    CONST robtarget p14641:= [[1510.9571216135703, 63.37345761549072, 1006.500033578516], [0, 0, 1, 0], [0, 0, 0, 0], [9E9, 9E9, 9E9, 9E9, 9E9, 9E9]];
    CONST robtarget p14642:= [[1511.1184630222722, 63.35487120853786, 1006.500033578516], [0, 0, 1, 0], [0, 0, 0, 0], [9E9, 9E9, 9E9, 9E9, 9E9, 9E9]];
    CONST robtarget p14643:= [[1511.1919380294153, 63.341381931287984, 1006.500033578516], [0, 0, 1, 0], [0, 0, 0, 0], [9E9, 9E9, 9E9, 9E9, 9E9, 9E9]];
    CONST robtarget p14644:= [[1512.026838057439, 63.17846774539392, 1006.500033578516], [0, 0, 1, 0], [0, 0, 0, 0], [9E9, 9E9, 9E9, 9E9, 9E9, 9E9]];
    CONST robtarget p14645:= [[1512.5585207158877, 63.05117882240624, 1006.500033578516], [0, 0, 1, 0], [0, 0, 0, 0], [9E9, 9E9, 9E9, 9E9, 9E9, 9E9]];
    CONST robtarget p14646:= [[1512.9152156348257, 62.99334195486536, 1006.500033578516], [0, 0, 1, 0], [0, 0, 0, 0], [9E9, 9E9, 9E9, 9E9, 9E9, 9E9]];
    CONST robtarget p14647:= [[1513.798506951844, 62.783709162407874, 1006.500033578516], [0, 0, 1, 0], [0, 0, 0, 0], [9E9, 9E9, 9E9, 9E9, 9E9, 9E9]];
    CONST robtarget p14648:= [[1514.847567863613, 62.563530246518, 1006.500033578516], [0, 0, 1, 0], [0, 0, 0, 0], [9E9, 9E9, 9E9, 9E9, 9E9, 9E9]];
    CONST robtarget p14649:= [[1515.255096833937, 62.462945925381334, 1006.500033578516], [0, 0, 1, 0], [0, 0, 0, 0], [9E9, 9E9, 9E9, 9E9, 9E9, 9E9]];
    CONST robtarget p14650:= [[1515.509041751135, 62.41476108124637, 1006.500033578516], [0, 0, 1, 0], [0, 0, 0, 0], [9E9, 9E9, 9E9, 9E9, 9E9, 9E9]];
    CONST robtarget p14651:= [[1515.8348657437182, 62.34037513585322, 1006.500033578516], [0, 0, 1, 0], [0, 0, 0, 0], [9E9, 9E9, 9E9, 9E9, 9E9, 9E9]];
    CONST robtarget p14652:= [[1516.3628032758625, 62.21258930958216, 1006.500033578516], [0, 0, 1, 0], [0, 0, 0, 0], [9E9, 9E9, 9E9, 9E9, 9E9, 9E9]];
    CONST robtarget p14653:= [[1516.8558086004887, 62.054342846622134, 1006.500033578516], [0, 0, 1, 0], [0, 0, 0, 0], [9E9, 9E9, 9E9, 9E9, 9E9, 9E9]];
    CONST robtarget p14654:= [[1516.94184995351, 62.01985911324756, 1006.500033578516], [0, 0, 1, 0], [0, 0, 0, 0], [9E9, 9E9, 9E9, 9E9, 9E9, 9E9]];
    CONST robtarget p14655:= [[1517.8260139593945, 61.7655492376807, 1006.500033578516], [0, 0, 1, 0], [0, 0, 0, 0], [9E9, 9E9, 9E9, 9E9, 9E9, 9E9]];
    CONST robtarget p14656:= [[1518.3959985979216, 61.59972849280017, 1006.500033578516], [0, 0, 1, 0], [0, 0, 0, 0], [9E9, 9E9, 9E9, 9E9, 9E9, 9E9]];
    CONST robtarget p14657:= [[1519.0877750129548, 61.40495027580202, 1006.500033578516], [0, 0, 1, 0], [0, 0, 0, 0], [9E9, 9E9, 9E9, 9E9, 9E9, 9E9]];
    CONST robtarget p14658:= [[1519.4220256911422, 61.30068815369448, 1006.500033578516], [0, 0, 1, 0], [0, 0, 0, 0], [9E9, 9E9, 9E9, 9E9, 9E9, 9E9]];
    CONST robtarget p14659:= [[1520.4546810078716, 60.9628761084728, 1006.500033578516], [0, 0, 1, 0], [0, 0, 0, 0], [9E9, 9E9, 9E9, 9E9, 9E9, 9E9]];
    CONST robtarget p14660:= [[1520.7208420853615, 60.899099294826286, 1006.500033578516], [0, 0, 1, 0], [0, 0, 0, 0], [9E9, 9E9, 9E9, 9E9, 9E9, 9E9]];
    CONST robtarget p14661:= [[1520.9944154401092, 60.79050565777585, 1006.500033578516], [0, 0, 1, 0], [0, 0, 0, 0], [9E9, 9E9, 9E9, 9E9, 9E9, 9E9]];
    CONST robtarget p14662:= [[1521.468460467742, 60.619702144143545, 1006.500033578516], [0, 0, 1, 0], [0, 0, 0, 0], [9E9, 9E9, 9E9, 9E9, 9E9, 9E9]];
    CONST robtarget p14663:= [[1522.0539891001142, 60.40291207086237, 1006.500033578516], [0, 0, 1, 0], [0, 0, 0, 0], [9E9, 9E9, 9E9, 9E9, 9E9, 9E9]];
    CONST robtarget p14664:= [[1522.7235250206843, 60.13765981750545, 1006.500033578516], [0, 0, 1, 0], [0, 0, 0, 0], [9E9, 9E9, 9E9, 9E9, 9E9, 9E9]];
    CONST robtarget p14665:= [[1522.7540810701935, 60.12646280502547, 1006.500033578516], [0, 0, 1, 0], [0, 0, 0, 0], [9E9, 9E9, 9E9, 9E9, 9E9, 9E9]];
    CONST robtarget p14666:= [[1522.977172790825, 60.0450909611216, 1006.500033578516], [0, 0, 1, 0], [0, 0, 0, 0], [9E9, 9E9, 9E9, 9E9, 9E9, 9E9]];
    CONST robtarget p14667:= [[1523.8573489774064, 59.71048583629785, 1006.500033578516], [0, 0, 1, 0], [0, 0, 0, 0], [9E9, 9E9, 9E9, 9E9, 9E9, 9E9]];
    CONST robtarget p14668:= [[1524.305158114966, 59.53535137429769, 1006.500033578516], [0, 0, 1, 0], [0, 0, 0, 0], [9E9, 9E9, 9E9, 9E9, 9E9, 9E9]];
    CONST robtarget p14669:= [[1524.656610079094, 59.40530950563833, 1006.500033578516], [0, 0, 1, 0], [0, 0, 0, 0], [9E9, 9E9, 9E9, 9E9, 9E9, 9E9]];
    CONST robtarget p14670:= [[1525.149298617828, 59.17779911458156, 1006.500033578516], [0, 0, 1, 0], [0, 0, 0, 0], [9E9, 9E9, 9E9, 9E9, 9E9, 9E9]];
    CONST robtarget p14671:= [[1525.7575127352557, 58.87613102467979, 1006.500033578516], [0, 0, 1, 0], [0, 0, 0, 0], [9E9, 9E9, 9E9, 9E9, 9E9, 9E9]];
    CONST robtarget p14672:= [[1526.170972481238, 58.714980753068446, 1006.500033578516], [0, 0, 1, 0], [0, 0, 0, 0], [9E9, 9E9, 9E9, 9E9, 9E9, 9E9]];
    CONST robtarget p14673:= [[1526.7257950856722, 58.46470075930664, 1006.500033578516], [0, 0, 1, 0], [0, 0, 0, 0], [9E9, 9E9, 9E9, 9E9, 9E9, 9E9]];
    CONST robtarget p14674:= [[1527.3077094242446, 58.20997178842184, 1006.500033578516], [0, 0, 1, 0], [0, 0, 0, 0], [9E9, 9E9, 9E9, 9E9, 9E9, 9E9]];
    CONST robtarget p14675:= [[1527.6845666037234, 58.0161366438124, 1006.500033578516], [0, 0, 1, 0], [0, 0, 0, 0], [9E9, 9E9, 9E9, 9E9, 9E9, 9E9]];
    CONST robtarget p14676:= [[1527.8326061398718, 57.948812745233525, 1006.500033578516], [0, 0, 1, 0], [0, 0, 0, 0], [9E9, 9E9, 9E9, 9E9, 9E9, 9E9]];
    CONST robtarget p14677:= [[1528.3321808852675, 57.69325378961487, 1006.500033578516], [0, 0, 1, 0], [0, 0, 0, 0], [9E9, 9E9, 9E9, 9E9, 9E9, 9E9]];
    CONST robtarget p14678:= [[1528.403927309375, 57.65748391653119, 1006.500033578516], [0, 0, 1, 0], [0, 0, 0, 0], [9E9, 9E9, 9E9, 9E9, 9E9, 9E9]];
    CONST robtarget p14679:= [[1528.9869187812067, 57.39394460057444, 1006.500033578516], [0, 0, 1, 0], [0, 0, 0, 0], [9E9, 9E9, 9E9, 9E9, 9E9, 9E9]];
    CONST robtarget p14680:= [[1529.2613805009244, 57.26779957940987, 1006.500033578516], [0, 0, 1, 0], [0, 0, 0, 0], [9E9, 9E9, 9E9, 9E9, 9E9, 9E9]];
    CONST robtarget p14681:= [[1529.6697738066682, 57.06843620345721, 1006.500033578516], [0, 0, 1, 0], [0, 0, 0, 0], [9E9, 9E9, 9E9, 9E9, 9E9, 9E9]];
    CONST robtarget p14682:= [[1530.2856563586133, 56.72445722365994, 1006.500033578516], [0, 0, 1, 0], [0, 0, 0, 0], [9E9, 9E9, 9E9, 9E9, 9E9, 9E9]];
    CONST robtarget p14683:= [[1530.8126991827496, 56.4341660345891, 1006.500033578516], [0, 0, 1, 0], [0, 0, 0, 0], [9E9, 9E9, 9E9, 9E9, 9E9, 9E9]];
    CONST robtarget p14684:= [[1530.9029259654756, 56.3783277374728, 1006.500033578516], [0, 0, 1, 0], [0, 0, 0, 0], [9E9, 9E9, 9E9, 9E9, 9E9, 9E9]];
    CONST robtarget p14685:= [[1531.0054963877374, 56.315172306385094, 1006.500033578516], [0, 0, 1, 0], [0, 0, 0, 0], [9E9, 9E9, 9E9, 9E9, 9E9, 9E9]];
    CONST robtarget p14686:= [[1531.3939612691959, 56.09683858981346, 1006.500033578516], [0, 0, 1, 0], [0, 0, 0, 0], [9E9, 9E9, 9E9, 9E9, 9E9, 9E9]];
    CONST robtarget p14687:= [[1531.8623727083182, 55.83685599433868, 1006.500033578516], [0, 0, 1, 0], [0, 0, 0, 0], [9E9, 9E9, 9E9, 9E9, 9E9, 9E9]];
    CONST robtarget p14688:= [[1532.024440070901, 55.73722495097826, 1006.500033578516], [0, 0, 1, 0], [0, 0, 0, 0], [9E9, 9E9, 9E9, 9E9, 9E9, 9E9]];
    CONST robtarget p14689:= [[1532.7201519563368, 55.36777082129741, 1006.500033578516], [0, 0, 1, 0], [0, 0, 0, 0], [9E9, 9E9, 9E9, 9E9, 9E9, 9E9]];
    CONST robtarget p14690:= [[1533.2451221887477, 55.05705588289027, 1006.500033578516], [0, 0, 1, 0], [0, 0, 0, 0], [9E9, 9E9, 9E9, 9E9, 9E9, 9E9]];
    CONST robtarget p14691:= [[1533.6846313226854, 54.805458357707266, 1006.500033578516], [0, 0, 1, 0], [0, 0, 0, 0], [9E9, 9E9, 9E9, 9E9, 9E9, 9E9]];
    CONST robtarget p14692:= [[1533.8934584959652, 54.65278530648348, 1006.500033578516], [0, 0, 1, 0], [0, 0, 0, 0], [9E9, 9E9, 9E9, 9E9, 9E9, 9E9]];
    CONST robtarget p14693:= [[1534.2116287991314, 54.4123880238884, 1006.500033578516], [0, 0, 1, 0], [0, 0, 0, 0], [9E9, 9E9, 9E9, 9E9, 9E9, 9E9]];
    CONST robtarget p14694:= [[1534.6901098946857, 54.118222023287345, 1006.500033578516], [0, 0, 1, 0], [0, 0, 0, 0], [9E9, 9E9, 9E9, 9E9, 9E9, 9E9]];
    CONST robtarget p14695:= [[1535.3882444304677, 53.67964368227618, 1006.500033578516], [0, 0, 1, 0], [0, 0, 0, 0], [9E9, 9E9, 9E9, 9E9, 9E9, 9E9]];
    CONST robtarget p14696:= [[1535.6440065674608, 53.48641652408345, 1006.500033578516], [0, 0, 1, 0], [0, 0, 0, 0], [9E9, 9E9, 9E9, 9E9, 9E9, 9E9]];
    CONST robtarget p14697:= [[1536.2093768314423, 53.097910660736204, 1006.500033578516], [0, 0, 1, 0], [0, 0, 0, 0], [9E9, 9E9, 9E9, 9E9, 9E9, 9E9]];
    CONST robtarget p14698:= [[1536.9779076559207, 52.624035474973724, 1006.500033578516], [0, 0, 1, 0], [0, 0, 0, 0], [9E9, 9E9, 9E9, 9E9, 9E9, 9E9]];
    CONST robtarget p14699:= [[1537.4393405989101, 52.32171516144058, 1006.500033578516], [0, 0, 1, 0], [0, 0, 0, 0], [9E9, 9E9, 9E9, 9E9, 9E9, 9E9]];
    CONST robtarget p14700:= [[1537.952006745379, 51.91517388024164, 1006.500033578516], [0, 0, 1, 0], [0, 0, 0, 0], [9E9, 9E9, 9E9, 9E9, 9E9, 9E9]];
    CONST robtarget p14701:= [[1538.2226229328674, 51.700360577582046, 1006.500033578516], [0, 0, 1, 0], [0, 0, 0, 0], [9E9, 9E9, 9E9, 9E9, 9E9, 9E9]];
    CONST robtarget p14702:= [[1538.5500075167402, 51.46408461899675, 1006.500033578516], [0, 0, 1, 0], [0, 0, 0, 0], [9E9, 9E9, 9E9, 9E9, 9E9, 9E9]];
    CONST robtarget p14703:= [[1538.9225032761597, 51.18184185491022, 1006.500033578516], [0, 0, 1, 0], [0, 0, 0, 0], [9E9, 9E9, 9E9, 9E9, 9E9, 9E9]];
    CONST robtarget p14704:= [[1539.2375324072243, 50.939131502791724, 1006.500033578516], [0, 0, 1, 0], [0, 0, 0, 0], [9E9, 9E9, 9E9, 9E9, 9E9, 9E9]];
    CONST robtarget p14705:= [[1540.1829191616407, 50.145246062498, 1006.500033578516], [0, 0, 1, 0], [0, 0, 0, 0], [9E9, 9E9, 9E9, 9E9, 9E9, 9E9]];
    CONST robtarget p14706:= [[1540.6342645888235, 49.82479613541888, 1006.500033578516], [0, 0, 1, 0], [0, 0, 0, 0], [9E9, 9E9, 9E9, 9E9, 9E9, 9E9]];
    CONST robtarget p14707:= [[1541.3997951640697, 49.20201413735353, 1006.500033578516], [0, 0, 1, 0], [0, 0, 0, 0], [9E9, 9E9, 9E9, 9E9, 9E9, 9E9]];
    CONST robtarget p14708:= [[1542.2802015710938, 48.44291913123219, 1006.500033578516], [0, 0, 1, 0], [0, 0, 0, 0], [9E9, 9E9, 9E9, 9E9, 9E9, 9E9]];
    CONST robtarget p14709:= [[1542.848436210057, 47.911154253194894, 1006.500033578516], [0, 0, 1, 0], [0, 0, 0, 0], [9E9, 9E9, 9E9, 9E9, 9E9, 9E9]];
    CONST robtarget p14710:= [[1543.249750681818, 47.58041096004163, 1006.500033578516], [0, 0, 1, 0], [0, 0, 0, 0], [9E9, 9E9, 9E9, 9E9, 9E9, 9E9]];
    CONST robtarget p14711:= [[1543.8613961148844, 46.98941101413523, 1006.500033578516], [0, 0, 1, 0], [0, 0, 0, 0], [9E9, 9E9, 9E9, 9E9, 9E9, 9E9]];
    CONST robtarget p14712:= [[1544.0446499071509, 46.83874137102008, 1006.500033578516], [0, 0, 1, 0], [0, 0, 0, 0], [9E9, 9E9, 9E9, 9E9, 9E9, 9E9]];
    CONST robtarget p14713:= [[1544.2953989022335, 46.61563060487386, 1006.500033578516], [0, 0, 1, 0], [0, 0, 0, 0], [9E9, 9E9, 9E9, 9E9, 9E9, 9E9]];
    CONST robtarget p14714:= [[1544.54804056772, 46.38574176255722, 1006.500033578516], [0, 0, 1, 0], [0, 0, 0, 0], [9E9, 9E9, 9E9, 9E9, 9E9, 9E9]];
    CONST robtarget p14715:= [[1544.635189922801, 46.31124549330636, 1006.500033578516], [0, 0, 1, 0], [0, 0, 0, 0], [9E9, 9E9, 9E9, 9E9, 9E9, 9E9]];
    CONST robtarget p14716:= [[1545.4540333634932, 45.48335179072561, 1006.500033578516], [0, 0, 1, 0], [0, 0, 0, 0], [9E9, 9E9, 9E9, 9E9, 9E9, 9E9]];
    CONST robtarget p14717:= [[1545.7644585194985, 45.10437831876281, 1006.500033578516], [0, 0, 1, 0], [0, 0, 0, 0], [9E9, 9E9, 9E9, 9E9, 9E9, 9E9]];
    CONST robtarget p14718:= [[1546.0127018950527, 44.843745114856446, 1006.500033578516], [0, 0, 1, 0], [0, 0, 0, 0], [9E9, 9E9, 9E9, 9E9, 9E9, 9E9]];
    CONST robtarget p14719:= [[1546.7740572911337, 44.03270232293215, 1006.500033578516], [0, 0, 1, 0], [0, 0, 0, 0], [9E9, 9E9, 9E9, 9E9, 9E9, 9E9]];
    CONST robtarget p14720:= [[1547.0970360263204, 43.759023791525095, 1006.500033578516], [0, 0, 1, 0], [0, 0, 0, 0], [9E9, 9E9, 9E9, 9E9, 9E9, 9E9]];
    CONST robtarget p14721:= [[1547.2985281571125, 43.556821645131976, 1006.500033578516], [0, 0, 1, 0], [0, 0, 0, 0], [9E9, 9E9, 9E9, 9E9, 9E9, 9E9]];
    CONST robtarget p14722:= [[1547.5784264326533, 43.24559099443002, 1006.500033578516], [0, 0, 1, 0], [0, 0, 0, 0], [9E9, 9E9, 9E9, 9E9, 9E9, 9E9]];
    CONST robtarget p14723:= [[1547.840639915275, 42.976910613143446, 1006.500033578516], [0, 0, 1, 0], [0, 0, 0, 0], [9E9, 9E9, 9E9, 9E9, 9E9, 9E9]];
    CONST robtarget p14724:= [[1548.5685814620201, 42.11718983212772, 1006.500033578516], [0, 0, 1, 0], [0, 0, 0, 0], [9E9, 9E9, 9E9, 9E9, 9E9, 9E9]];
    CONST robtarget p14725:= [[1549.0589016644108, 41.54224515009723, 1006.500033578516], [0, 0, 1, 0], [0, 0, 0, 0], [9E9, 9E9, 9E9, 9E9, 9E9, 9E9]];
    CONST robtarget p14726:= [[1549.1397925073998, 41.45436251768466, 1006.500033578516], [0, 0, 1, 0], [0, 0, 0, 0], [9E9, 9E9, 9E9, 9E9, 9E9, 9E9]];
    CONST robtarget p14727:= [[1549.3841406789884, 41.1427679591735, 1006.500033578516], [0, 0, 1, 0], [0, 0, 0, 0], [9E9, 9E9, 9E9, 9E9, 9E9, 9E9]];
    CONST robtarget p14728:= [[1549.5239794339052, 40.95950274767945, 1006.500033578516], [0, 0, 1, 0], [0, 0, 0, 0], [9E9, 9E9, 9E9, 9E9, 9E9, 9E9]];
    CONST robtarget p14729:= [[1549.9175539397738, 40.51438406992901, 1006.500033578516], [0, 0, 1, 0], [0, 0, 0, 0], [9E9, 9E9, 9E9, 9E9, 9E9, 9E9]];
    CONST robtarget p14730:= [[1550.3216633796537, 40.038823451018516, 1006.500033578516], [0, 0, 1, 0], [0, 0, 0, 0], [9E9, 9E9, 9E9, 9E9, 9E9, 9E9]];
    CONST robtarget p14731:= [[1550.4495787903381, 39.860864577949286, 1006.500033578516], [0, 0, 1, 0], [0, 0, 0, 0], [9E9, 9E9, 9E9, 9E9, 9E9, 9E9]];
    CONST robtarget p14732:= [[1550.6937743751787, 39.5427168649649, 1006.500033578516], [0, 0, 1, 0], [0, 0, 0, 0], [9E9, 9E9, 9E9, 9E9, 9E9, 9E9]];
    CONST robtarget p14733:= [[1551.2596416418764, 38.84732865927106, 1006.500033578516], [0, 0, 1, 0], [0, 0, 0, 0], [9E9, 9E9, 9E9, 9E9, 9E9, 9E9]];
    CONST robtarget p14734:= [[1551.6870753715048, 38.25053385446556, 1006.500033578516], [0, 0, 1, 0], [0, 0, 0, 0], [9E9, 9E9, 9E9, 9E9, 9E9, 9E9]];
    CONST robtarget p14735:= [[1551.8361490020857, 38.01625032551375, 1006.500033578516], [0, 0, 1, 0], [0, 0, 0, 0], [9E9, 9E9, 9E9, 9E9, 9E9, 9E9]];
    CONST robtarget p14736:= [[1552.322823514699, 37.36153510210862, 1006.500033578516], [0, 0, 1, 0], [0, 0, 0, 0], [9E9, 9E9, 9E9, 9E9, 9E9, 9E9]];
    CONST robtarget p14737:= [[1552.5842476544994, 36.958893981652636, 1006.500033578516], [0, 0, 1, 0], [0, 0, 0, 0], [9E9, 9E9, 9E9, 9E9, 9E9, 9E9]];
    CONST robtarget p14738:= [[1552.8616551509776, 36.5874901381969, 1006.500033578516], [0, 0, 1, 0], [0, 0, 0, 0], [9E9, 9E9, 9E9, 9E9, 9E9, 9E9]];
    CONST robtarget p14739:= [[1553.159967137924, 36.201259725787494, 1006.500033578516], [0, 0, 1, 0], [0, 0, 0, 0], [9E9, 9E9, 9E9, 9E9, 9E9, 9E9]];
    CONST robtarget p14740:= [[1553.3919006865265, 35.845938138459914, 1006.500033578516], [0, 0, 1, 0], [0, 0, 0, 0], [9E9, 9E9, 9E9, 9E9, 9E9, 9E9]];
    CONST robtarget p14741:= [[1553.4492538776192, 35.75324229238505, 1006.500033578516], [0, 0, 1, 0], [0, 0, 0, 0], [9E9, 9E9, 9E9, 9E9, 9E9, 9E9]];
    CONST robtarget p14742:= [[1553.6849733642457, 35.35776058704826, 1006.500033578516], [0, 0, 1, 0], [0, 0, 0, 0], [9E9, 9E9, 9E9, 9E9, 9E9, 9E9]];
    CONST robtarget p14743:= [[1554.0221492244746, 34.890455488715006, 1006.500033578516], [0, 0, 1, 0], [0, 0, 0, 0], [9E9, 9E9, 9E9, 9E9, 9E9, 9E9]];
    CONST robtarget p14744:= [[1554.3819330409094, 34.311998246707276, 1006.500033578516], [0, 0, 1, 0], [0, 0, 0, 0], [9E9, 9E9, 9E9, 9E9, 9E9, 9E9]];
    CONST robtarget p14745:= [[1554.7324883746796, 33.72360383375208, 1006.500033578516], [0, 0, 1, 0], [0, 0, 0, 0], [9E9, 9E9, 9E9, 9E9, 9E9, 9E9]];
    CONST robtarget p14746:= [[1554.9694331765027, 33.34150920841043, 1006.500033578516], [0, 0, 1, 0], [0, 0, 0, 0], [9E9, 9E9, 9E9, 9E9, 9E9, 9E9]];
    CONST robtarget p14747:= [[1555.0578363454322, 33.18808941710759, 1006.500033578516], [0, 0, 1, 0], [0, 0, 0, 0], [9E9, 9E9, 9E9, 9E9, 9E9, 9E9]];
    CONST robtarget p14748:= [[1555.5191903887774, 32.347242553330574, 1006.500033578516], [0, 0, 1, 0], [0, 0, 0, 0], [9E9, 9E9, 9E9, 9E9, 9E9, 9E9]];
    CONST robtarget p14749:= [[1555.899208185482, 31.751166868234478, 1006.500033578516], [0, 0, 1, 0], [0, 0, 0, 0], [9E9, 9E9, 9E9, 9E9, 9E9, 9E9]];
    CONST robtarget p14750:= [[1556.105965761014, 31.457408539315693, 1006.500033578516], [0, 0, 1, 0], [0, 0, 0, 0], [9E9, 9E9, 9E9, 9E9, 9E9, 9E9]];
    CONST robtarget p14751:= [[1556.2761023181502, 31.162061354166894, 1006.500033578516], [0, 0, 1, 0], [0, 0, 0, 0], [9E9, 9E9, 9E9, 9E9, 9E9, 9E9]];
    CONST robtarget p14752:= [[1556.420299300182, 30.87457089103094, 1006.500033578516], [0, 0, 1, 0], [0, 0, 0, 0], [9E9, 9E9, 9E9, 9E9, 9E9, 9E9]];
    CONST robtarget p14753:= [[1556.6192652398609, 30.460695675097654, 1006.500033578516], [0, 0, 1, 0], [0, 0, 0, 0], [9E9, 9E9, 9E9, 9E9, 9E9, 9E9]];
    CONST robtarget p14754:= [[1556.8508635062612, 29.96949114767618, 1006.500033578516], [0, 0, 1, 0], [0, 0, 0, 0], [9E9, 9E9, 9E9, 9E9, 9E9, 9E9]];
    CONST robtarget p14755:= [[1557.0508965859028, 29.617423973888137, 1006.500033578516], [0, 0, 1, 0], [0, 0, 0, 0], [9E9, 9E9, 9E9, 9E9, 9E9, 9E9]];
    CONST robtarget p14756:= [[1557.4062954918465, 28.908772989595676, 1006.500033578516], [0, 0, 1, 0], [0, 0, 0, 0], [9E9, 9E9, 9E9, 9E9, 9E9, 9E9]];
    CONST robtarget p14757:= [[1557.591791517242, 28.580906463463975, 1006.500033578516], [0, 0, 1, 0], [0, 0, 0, 0], [9E9, 9E9, 9E9, 9E9, 9E9, 9E9]];
    CONST robtarget p14758:= [[1558.0102406682965, 27.771073474515347, 1006.500033578516], [0, 0, 1, 0], [0, 0, 0, 0], [9E9, 9E9, 9E9, 9E9, 9E9, 9E9]];
    CONST robtarget p14759:= [[1558.5100146038824, 26.696173383688503, 1006.500033578516], [0, 0, 1, 0], [0, 0, 0, 0], [9E9, 9E9, 9E9, 9E9, 9E9, 9E9]];
    CONST robtarget p14760:= [[1558.6483628452322, 26.346591876591773, 1006.500033578516], [0, 0, 1, 0], [0, 0, 0, 0], [9E9, 9E9, 9E9, 9E9, 9E9, 9E9]];
    CONST robtarget p14761:= [[1558.9049415700476, 25.77297683860722, 1006.500033578516], [0, 0, 1, 0], [0, 0, 0, 0], [9E9, 9E9, 9E9, 9E9, 9E9, 9E9]];
    CONST robtarget p14762:= [[1559.1828014244882, 25.12800186908713, 1006.500033578516], [0, 0, 1, 0], [0, 0, 0, 0], [9E9, 9E9, 9E9, 9E9, 9E9, 9E9]];
    CONST robtarget p14763:= [[1559.3533095895443, 24.673409310394717, 1006.500033578516], [0, 0, 1, 0], [0, 0, 0, 0], [9E9, 9E9, 9E9, 9E9, 9E9, 9E9]];
    CONST robtarget p14764:= [[1559.5848736434261, 24.07845287627731, 1006.500033578516], [0, 0, 1, 0], [0, 0, 0, 0], [9E9, 9E9, 9E9, 9E9, 9E9, 9E9]];
    CONST robtarget p14765:= [[1559.813760776618, 23.638280641204958, 1006.500033578516], [0, 0, 1, 0], [0, 0, 0, 0], [9E9, 9E9, 9E9, 9E9, 9E9, 9E9]];
    CONST robtarget p14766:= [[1560.0305384185972, 23.07452224167156, 1006.500033578516], [0, 0, 1, 0], [0, 0, 0, 0], [9E9, 9E9, 9E9, 9E9, 9E9, 9E9]];
    CONST robtarget p14767:= [[1560.1435635645735, 22.84049973394798, 1006.500033578516], [0, 0, 1, 0], [0, 0, 0, 0], [9E9, 9E9, 9E9, 9E9, 9E9, 9E9]];
    CONST robtarget p14768:= [[1560.226070512941, 22.531314308390435, 1006.500033578516], [0, 0, 1, 0], [0, 0, 0, 0], [9E9, 9E9, 9E9, 9E9, 9E9, 9E9]];
    CONST robtarget p14769:= [[1560.2753114760053, 22.345030427414173, 1006.500033578516], [0, 0, 1, 0], [0, 0, 0, 0], [9E9, 9E9, 9E9, 9E9, 9E9, 9E9]];
    CONST robtarget p14770:= [[1560.5735676394168, 21.54628752008709, 1006.500033578516], [0, 0, 1, 0], [0, 0, 0, 0], [9E9, 9E9, 9E9, 9E9, 9E9, 9E9]];
    CONST robtarget p14771:= [[1560.5865985779046, 21.51311816527128, 1006.500033578516], [0, 0, 1, 0], [0, 0, 0, 0], [9E9, 9E9, 9E9, 9E9, 9E9, 9E9]];
    CONST robtarget p14772:= [[1560.7155063343944, 21.100773229791002, 1006.500033578516], [0, 0, 1, 0], [0, 0, 0, 0], [9E9, 9E9, 9E9, 9E9, 9E9, 9E9]];
    CONST robtarget p14773:= [[1560.8442825601521, 20.737343741796437, 1006.500033578516], [0, 0, 1, 0], [0, 0, 0, 0], [9E9, 9E9, 9E9, 9E9, 9E9, 9E9]];
    CONST robtarget p14774:= [[1560.8976160111743, 20.563431226153043, 1006.500033578516], [0, 0, 1, 0], [0, 0, 0, 0], [9E9, 9E9, 9E9, 9E9, 9E9, 9E9]];
    CONST robtarget p14775:= [[1561.2177020383199, 19.630147089741726, 1006.500033578516], [0, 0, 1, 0], [0, 0, 0, 0], [9E9, 9E9, 9E9, 9E9, 9E9, 9E9]];
    CONST robtarget p14776:= [[1561.4639275811087, 18.912693395775676, 1006.500033578516], [0, 0, 1, 0], [0, 0, 0, 0], [9E9, 9E9, 9E9, 9E9, 9E9, 9E9]];
    CONST robtarget p14777:= [[1561.6583606547026, 18.321669832533203, 1006.500033578516], [0, 0, 1, 0], [0, 0, 0, 0], [9E9, 9E9, 9E9, 9E9, 9E9, 9E9]];
    CONST robtarget p14778:= [[1561.7259002676185, 18.087761559197332, 1006.500033578516], [0, 0, 1, 0], [0, 0, 0, 0], [9E9, 9E9, 9E9, 9E9, 9E9, 9E9]];
    CONST robtarget p14779:= [[1561.9203310868406, 17.29266482364558, 1006.500033578516], [0, 0, 1, 0], [0, 0, 0, 0], [9E9, 9E9, 9E9, 9E9, 9E9, 9E9]];
    CONST robtarget p14780:= [[1561.9773013858805, 17.06323004336498, 1006.500033578516], [0, 0, 1, 0], [0, 0, 0, 0], [9E9, 9E9, 9E9, 9E9, 9E9, 9E9]];
    CONST robtarget p14781:= [[1562.1756853904667, 16.355823136074605, 1006.500033578516], [0, 0, 1, 0], [0, 0, 0, 0], [9E9, 9E9, 9E9, 9E9, 9E9, 9E9]];
    CONST robtarget p14782:= [[1562.3204272341718, 15.699428292366264, 1006.500033578516], [0, 0, 1, 0], [0, 0, 0, 0], [9E9, 9E9, 9E9, 9E9, 9E9, 9E9]];
    CONST robtarget p14783:= [[1562.5445745281302, 14.740266897005455, 1006.500033578516], [0, 0, 1, 0], [0, 0, 0, 0], [9E9, 9E9, 9E9, 9E9, 9E9, 9E9]];
    CONST robtarget p14784:= [[1562.675887940053, 14.34057446811299, 1006.500033578516], [0, 0, 1, 0], [0, 0, 0, 0], [9E9, 9E9, 9E9, 9E9, 9E9, 9E9]];
    CONST robtarget p14785:= [[1562.8223840780483, 13.760772988322543, 1006.500033578516], [0, 0, 1, 0], [0, 0, 0, 0], [9E9, 9E9, 9E9, 9E9, 9E9, 9E9]];
    CONST robtarget p14786:= [[1562.901529968312, 13.355693959034014, 1006.500033578516], [0, 0, 1, 0], [0, 0, 0, 0], [9E9, 9E9, 9E9, 9E9, 9E9, 9E9]];
    CONST robtarget p14787:= [[1563.0528539818283, 12.52897697257535, 1006.500033578516], [0, 0, 1, 0], [0, 0, 0, 0], [9E9, 9E9, 9E9, 9E9, 9E9, 9E9]];
    CONST robtarget p14788:= [[1563.1557063470802, 12.054831410101713, 1006.500033578516], [0, 0, 1, 0], [0, 0, 0, 0], [9E9, 9E9, 9E9, 9E9, 9E9, 9E9]];
    CONST robtarget p14789:= [[1563.2423103824246, 11.479109892409923, 1006.500033578516], [0, 0, 1, 0], [0, 0, 0, 0], [9E9, 9E9, 9E9, 9E9, 9E9, 9E9]];
    CONST robtarget p14790:= [[1563.266286273107, 11.342432296307521, 1006.500033578516], [0, 0, 1, 0], [0, 0, 0, 0], [9E9, 9E9, 9E9, 9E9, 9E9, 9E9]];
    CONST robtarget p14791:= [[1563.452496210667, 10.393351643055098, 1006.500033578516], [0, 0, 1, 0], [0, 0, 0, 0], [9E9, 9E9, 9E9, 9E9, 9E9, 9E9]];
    CONST robtarget p14792:= [[1563.5751833217294, 9.791225223977278, 1006.500033578516], [0, 0, 1, 0], [0, 0, 0, 0], [9E9, 9E9, 9E9, 9E9, 9E9, 9E9]];
    CONST robtarget p14793:= [[1563.641005792793, 9.41225053732255, 1006.500033578516], [0, 0, 1, 0], [0, 0, 0, 0], [9E9, 9E9, 9E9, 9E9, 9E9, 9E9]];
    CONST robtarget p14794:= [[1563.7037032071917, 8.785713771097988, 1006.500033578516], [0, 0, 1, 0], [0, 0, 0, 0], [9E9, 9E9, 9E9, 9E9, 9E9, 9E9]];
    CONST robtarget p14795:= [[1563.7468492957848, 8.295771319404253, 1006.500033578516], [0, 0, 1, 0], [0, 0, 0, 0], [9E9, 9E9, 9E9, 9E9, 9E9, 9E9]];
    CONST robtarget p14796:= [[1563.8508213879286, 7.462516168949108, 1006.500033578516], [0, 0, 1, 0], [0, 0, 0, 0], [9E9, 9E9, 9E9, 9E9, 9E9, 9E9]];
    CONST robtarget p14797:= [[1563.8869342178375, 7.130475393375889, 1006.500033578516], [0, 0, 1, 0], [0, 0, 0, 0], [9E9, 9E9, 9E9, 9E9, 9E9, 9E9]];
    CONST robtarget p14798:= [[1563.9039865967668, 6.677521872138911, 1006.500033578516], [0, 0, 1, 0], [0, 0, 0, 0], [9E9, 9E9, 9E9, 9E9, 9E9, 9E9]];
    CONST robtarget p14799:= [[1563.909465519574, 6.528256360088321, 1006.500033578516], [0, 0, 1, 0], [0, 0, 0, 0], [9E9, 9E9, 9E9, 9E9, 9E9, 9E9]];
    CONST robtarget p14800:= [[1564.060402070545, 5.411413458722052, 1006.500033578516], [0, 0, 1, 0], [0, 0, 0, 0], [9E9, 9E9, 9E9, 9E9, 9E9, 9E9]];
    CONST robtarget p14801:= [[1564.1523037088139, 4.7873673098910245, 1006.500033578516], [0, 0, 1, 0], [0, 0, 0, 0], [9E9, 9E9, 9E9, 9E9, 9E9, 9E9]];
    CONST robtarget p14802:= [[1564.1618904652082, 4.415172926905882, 1006.500033578516], [0, 0, 1, 0], [0, 0, 0, 0], [9E9, 9E9, 9E9, 9E9, 9E9, 9E9]];
    CONST robtarget p14803:= [[1564.193874845729, 3.6340002058411613, 1006.500033578516], [0, 0, 1, 0], [0, 0, 0, 0], [9E9, 9E9, 9E9, 9E9, 9E9, 9E9]];
    CONST robtarget p14804:= [[1564.208625048866, 3.306454787168562, 1006.500033578516], [0, 0, 1, 0], [0, 0, 0, 0], [9E9, 9E9, 9E9, 9E9, 9E9, 9E9]];
    CONST robtarget p14805:= [[1564.2216853064995, 2.6655686248283246, 1006.500033578516], [0, 0, 1, 0], [0, 0, 0, 0], [9E9, 9E9, 9E9, 9E9, 9E9, 9E9]];
    CONST robtarget p14806:= [[1564.256421588998, 2.2594512266854707, 1006.500033578516], [0, 0, 1, 0], [0, 0, 0, 0], [9E9, 9E9, 9E9, 9E9, 9E9, 9E9]];
    CONST robtarget p14807:= [[1564.3000812568512, 0.7193519216560702, 1006.500033578516], [0, 0, 1, 0], [0, 0, 0, 0], [9E9, 9E9, 9E9, 9E9, 9E9, 9E9]];
    CONST robtarget p14808:= [[1564.3361227675541, -0.026766125700305565, 1006.500033578516], [0, 0, 1, 0], [0, 0, 0, 0], [9E9, 9E9, 9E9, 9E9, 9E9, 9E9]];
    CONST robtarget p14809:= [[1564.30034650847, -0.9979191834767676, 1006.500033578516], [0, 0, 1, 0], [0, 0, 0, 0], [9E9, 9E9, 9E9, 9E9, 9E9, 9E9]];
    CONST robtarget p14810:= [[1564.2902268754742, -1.3355803424250183, 1006.500033578516], [0, 0, 1, 0], [0, 0, 0, 0], [9E9, 9E9, 9E9, 9E9, 9E9, 9E9]];
    CONST robtarget p14811:= [[1564.2395500118284, -1.9103519045936252, 1006.500033578516], [0, 0, 1, 0], [0, 0, 0, 0], [9E9, 9E9, 9E9, 9E9, 9E9, 9E9]];
    CONST robtarget p14812:= [[1564.224236137066, -2.6197755144861645, 1006.500033578516], [0, 0, 1, 0], [0, 0, 0, 0], [9E9, 9E9, 9E9, 9E9, 9E9, 9E9]];
    CONST robtarget p14813:= [[1564.2240335827769, -2.9068482163602454, 1006.500033578516], [0, 0, 1, 0], [0, 0, 0, 0], [9E9, 9E9, 9E9, 9E9, 9E9, 9E9]];
    CONST robtarget p14814:= [[1564.194042641247, -3.824350553576082, 1006.500033578516], [0, 0, 1, 0], [0, 0, 0, 0], [9E9, 9E9, 9E9, 9E9, 9E9, 9E9]];
    CONST robtarget p14815:= [[1564.1705646667035, -4.461289976446309, 1006.500033578516], [0, 0, 1, 0], [0, 0, 0, 0], [9E9, 9E9, 9E9, 9E9, 9E9, 9E9]];
    CONST robtarget p14816:= [[1564.0993585862266, -5.037353485207774, 1006.500033578516], [0, 0, 1, 0], [0, 0, 0, 0], [9E9, 9E9, 9E9, 9E9, 9E9, 9E9]];
    CONST robtarget p14817:= [[1564.0778761566255, -5.295004163286691, 1006.500033578516], [0, 0, 1, 0], [0, 0, 0, 0], [9E9, 9E9, 9E9, 9E9, 9E9, 9E9]];
    CONST robtarget p14818:= [[1564.0507910955898, -5.6657430795914365, 1006.500033578516], [0, 0, 1, 0], [0, 0, 0, 0], [9E9, 9E9, 9E9, 9E9, 9E9, 9E9]];
    CONST robtarget p14819:= [[1564.0362103933392, -5.891590708388563, 1006.500033578516], [0, 0, 1, 0], [0, 0, 0, 0], [9E9, 9E9, 9E9, 9E9, 9E9, 9E9]];
    CONST robtarget p14820:= [[1563.9578252628846, -6.483719773496958, 1006.500033578516], [0, 0, 1, 0], [0, 0, 0, 0], [9E9, 9E9, 9E9, 9E9, 9E9, 9E9]];
    CONST robtarget p14821:= [[1563.9140500083583, -6.806517664859392, 1006.500033578516], [0, 0, 1, 0], [0, 0, 0, 0], [9E9, 9E9, 9E9, 9E9, 9E9, 9E9]];
    CONST robtarget p14822:= [[1563.85314041922, -7.530970479438487, 1006.500033578516], [0, 0, 1, 0], [0, 0, 0, 0], [9E9, 9E9, 9E9, 9E9, 9E9, 9E9]];
    CONST robtarget p14823:= [[1563.7426549534343, -8.550826428317464, 1006.500033578516], [0, 0, 1, 0], [0, 0, 0, 0], [9E9, 9E9, 9E9, 9E9, 9E9, 9E9]];
    CONST robtarget p14824:= [[1563.7022531625055, -8.862064638755754, 1006.500033578516], [0, 0, 1, 0], [0, 0, 0, 0], [9E9, 9E9, 9E9, 9E9, 9E9, 9E9]];
    CONST robtarget p14825:= [[1563.6523033005042, -9.191708342134845, 1006.500033578516], [0, 0, 1, 0], [0, 0, 0, 0], [9E9, 9E9, 9E9, 9E9, 9E9, 9E9]];
    CONST robtarget p14826:= [[1563.5606913062238, -9.700379830138054, 1006.500033578516], [0, 0, 1, 0], [0, 0, 0, 0], [9E9, 9E9, 9E9, 9E9, 9E9, 9E9]];
    CONST robtarget p14827:= [[1563.501388077794, -10.062608269307404, 1006.500033578516], [0, 0, 1, 0], [0, 0, 0, 0], [9E9, 9E9, 9E9, 9E9, 9E9, 9E9]];
    CONST robtarget p14828:= [[1563.2958016283183, -11.040575674015209, 1006.500033578516], [0, 0, 1, 0], [0, 0, 0, 0], [9E9, 9E9, 9E9, 9E9, 9E9, 9E9]];
    CONST robtarget p14829:= [[1563.2338861768771, -11.53619279586249, 1006.500033578516], [0, 0, 1, 0], [0, 0, 0, 0], [9E9, 9E9, 9E9, 9E9, 9E9, 9E9]];
    CONST robtarget p14830:= [[1563.2110899575441, -11.66692031715386, 1006.500033578516], [0, 0, 1, 0], [0, 0, 0, 0], [9E9, 9E9, 9E9, 9E9, 9E9, 9E9]];
    CONST robtarget p14831:= [[1563.0576222911027, -12.4926757795307, 1006.500033578516], [0, 0, 1, 0], [0, 0, 0, 0], [9E9, 9E9, 9E9, 9E9, 9E9, 9E9]];
    CONST robtarget p14832:= [[1563.0027812761173, -12.79404840140765, 1006.500033578516], [0, 0, 1, 0], [0, 0, 0, 0], [9E9, 9E9, 9E9, 9E9, 9E9, 9E9]];
    CONST robtarget p14833:= [[1562.961957604833, -13.022518780506687, 1006.500033578516], [0, 0, 1, 0], [0, 0, 0, 0], [9E9, 9E9, 9E9, 9E9, 9E9, 9E9]];
    CONST robtarget p14834:= [[1562.868931608693, -13.41494549965634, 1006.500033578516], [0, 0, 1, 0], [0, 0, 0, 0], [9E9, 9E9, 9E9, 9E9, 9E9, 9E9]];
    CONST robtarget p14835:= [[1562.6114647241368, -14.68422796993785, 1006.500033578516], [0, 0, 1, 0], [0, 0, 0, 0], [9E9, 9E9, 9E9, 9E9, 9E9, 9E9]];
    CONST robtarget p14836:= [[1562.5993448072397, -14.75395399884816, 1006.500033578516], [0, 0, 1, 0], [0, 0, 0, 0], [9E9, 9E9, 9E9, 9E9, 9E9, 9E9]];
    CONST robtarget p14837:= [[1562.5695087422002, -14.868129949294513, 1006.500033578516], [0, 0, 1, 0], [0, 0, 0, 0], [9E9, 9E9, 9E9, 9E9, 9E9, 9E9]];
    CONST robtarget p14838:= [[1562.4621287233745, -15.23856788646195, 1006.500033578516], [0, 0, 1, 0], [0, 0, 0, 0], [9E9, 9E9, 9E9, 9E9, 9E9, 9E9]];
    CONST robtarget p14839:= [[1562.3134426502186, -15.812113512114948, 1006.500033578516], [0, 0, 1, 0], [0, 0, 0, 0], [9E9, 9E9, 9E9, 9E9, 9E9, 9E9]];
    CONST robtarget p14840:= [[1562.268086009388, -15.987293902563813, 1006.500033578516], [0, 0, 1, 0], [0, 0, 0, 0], [9E9, 9E9, 9E9, 9E9, 9E9, 9E9]];
    CONST robtarget p14841:= [[1562.0498727089093, -16.85698105824165, 1006.500033578516], [0, 0, 1, 0], [0, 0, 0, 0], [9E9, 9E9, 9E9, 9E9, 9E9, 9E9]];
    CONST robtarget p14842:= [[1561.868603398547, -17.404189316308575, 1006.500033578516], [0, 0, 1, 0], [0, 0, 0, 0], [9E9, 9E9, 9E9, 9E9, 9E9, 9E9]];
    CONST robtarget p14843:= [[1561.7089536960207, -18.046285020662488, 1006.500033578516], [0, 0, 1, 0], [0, 0, 0, 0], [9E9, 9E9, 9E9, 9E9, 9E9, 9E9]];
    CONST robtarget p14844:= [[1561.6434935010443, -18.380341739135275, 1006.500033578516], [0, 0, 1, 0], [0, 0, 0, 0], [9E9, 9E9, 9E9, 9E9, 9E9, 9E9]];
    CONST robtarget p14845:= [[1561.4980251653103, -18.801402093689738, 1006.500033578516], [0, 0, 1, 0], [0, 0, 0, 0], [9E9, 9E9, 9E9, 9E9, 9E9, 9E9]];
    CONST robtarget p14846:= [[1561.4025561047272, -19.134922793102973, 1006.500033578516], [0, 0, 1, 0], [0, 0, 0, 0], [9E9, 9E9, 9E9, 9E9, 9E9, 9E9]];
    CONST robtarget p14847:= [[1561.2476782256463, -19.598503249260126, 1006.500033578516], [0, 0, 1, 0], [0, 0, 0, 0], [9E9, 9E9, 9E9, 9E9, 9E9, 9E9]];
    CONST robtarget p14848:= [[1561.1058259162128, -20.009974983252526, 1006.500033578516], [0, 0, 1, 0], [0, 0, 0, 0], [9E9, 9E9, 9E9, 9E9, 9E9, 9E9]];
    CONST robtarget p14849:= [[1561.0179225265138, -20.231178944146002, 1006.500033578516], [0, 0, 1, 0], [0, 0, 0, 0], [9E9, 9E9, 9E9, 9E9, 9E9, 9E9]];
    CONST robtarget p14850:= [[1560.92544874012, -20.49418707914799, 1006.500033578516], [0, 0, 1, 0], [0, 0, 0, 0], [9E9, 9E9, 9E9, 9E9, 9E9, 9E9]];
    CONST robtarget p14851:= [[1560.7582369506374, -20.9658891268746, 1006.500033578516], [0, 0, 1, 0], [0, 0, 0, 0], [9E9, 9E9, 9E9, 9E9, 9E9, 9E9]];
    CONST robtarget p14852:= [[1560.4507217593277, -21.929743152602086, 1006.500033578516], [0, 0, 1, 0], [0, 0, 0, 0], [9E9, 9E9, 9E9, 9E9, 9E9, 9E9]];
    CONST robtarget p14853:= [[1560.2604531039328, -22.472044583540693, 1006.500033578516], [0, 0, 1, 0], [0, 0, 0, 0], [9E9, 9E9, 9E9, 9E9, 9E9, 9E9]];
    CONST robtarget p14854:= [[1560.0589552937367, -22.909557732998906, 1006.500033578516], [0, 0, 1, 0], [0, 0, 0, 0], [9E9, 9E9, 9E9, 9E9, 9E9, 9E9]];
    CONST robtarget p14855:= [[1559.6032390900743, -24.035680288262, 1006.500033578516], [0, 0, 1, 0], [0, 0, 0, 0], [9E9, 9E9, 9E9, 9E9, 9E9, 9E9]];
    CONST robtarget p14856:= [[1559.5326262761419, -24.271337139539995, 1006.500033578516], [0, 0, 1, 0], [0, 0, 0, 0], [9E9, 9E9, 9E9, 9E9, 9E9, 9E9]];
    CONST robtarget p14857:= [[1559.3901794184505, -24.619784221940208, 1006.500033578516], [0, 0, 1, 0], [0, 0, 0, 0], [9E9, 9E9, 9E9, 9E9, 9E9, 9E9]];
    CONST robtarget p14858:= [[1559.0194780159272, -25.393886851807324, 1006.500033578516], [0, 0, 1, 0], [0, 0, 0, 0], [9E9, 9E9, 9E9, 9E9, 9E9, 9E9]];
    CONST robtarget p14859:= [[1558.890902848407, -25.686679951722567, 1006.500033578516], [0, 0, 1, 0], [0, 0, 0, 0], [9E9, 9E9, 9E9, 9E9, 9E9, 9E9]];
    CONST robtarget p14860:= [[1558.7251377789137, -26.059862035002617, 1006.500033578516], [0, 0, 1, 0], [0, 0, 0, 0], [9E9, 9E9, 9E9, 9E9, 9E9, 9E9]];
    CONST robtarget p14861:= [[1558.5881050274124, -26.430467869774546, 1006.500033578516], [0, 0, 1, 0], [0, 0, 0, 0], [9E9, 9E9, 9E9, 9E9, 9E9, 9E9]];
    CONST robtarget p14862:= [[1558.1692143112832, -27.441466377842346, 1006.500033578516], [0, 0, 1, 0], [0, 0, 0, 0], [9E9, 9E9, 9E9, 9E9, 9E9, 9E9]];
    CONST robtarget p14863:= [[1558.1182924139741, -27.557330324648113, 1006.500033578516], [0, 0, 1, 0], [0, 0, 0, 0], [9E9, 9E9, 9E9, 9E9, 9E9, 9E9]];
    CONST robtarget p14864:= [[1557.7502894168094, -28.291309466763707, 1006.500033578516], [0, 0, 1, 0], [0, 0, 0, 0], [9E9, 9E9, 9E9, 9E9, 9E9, 9E9]];
    CONST robtarget p14865:= [[1557.5674734797851, -28.650617756356553, 1006.500033578516], [0, 0, 1, 0], [0, 0, 0, 0], [9E9, 9E9, 9E9, 9E9, 9E9, 9E9]];
    CONST robtarget p14866:= [[1557.3072447813986, -29.138133016690325, 1006.500033578516], [0, 0, 1, 0], [0, 0, 0, 0], [9E9, 9E9, 9E9, 9E9, 9E9, 9E9]];
    CONST robtarget p14867:= [[1557.2084248783242, -29.336507678844853, 1006.500033578516], [0, 0, 1, 0], [0, 0, 0, 0], [9E9, 9E9, 9E9, 9E9, 9E9, 9E9]];
    CONST robtarget p14868:= [[1557.1701662462808, -29.41181414533707, 1006.500033578516], [0, 0, 1, 0], [0, 0, 0, 0], [9E9, 9E9, 9E9, 9E9, 9E9, 9E9]];
    CONST robtarget p14869:= [[1556.752525535656, -30.173033556345423, 1006.500033578516], [0, 0, 1, 0], [0, 0, 0, 0], [9E9, 9E9, 9E9, 9E9, 9E9, 9E9]];
    CONST robtarget p14870:= [[1556.4193570309872, -30.844722309745045, 1006.500033578516], [0, 0, 1, 0], [0, 0, 0, 0], [9E9, 9E9, 9E9, 9E9, 9E9, 9E9]];
    CONST robtarget p14871:= [[1556.1364829738052, -31.358148580765054, 1006.500033578516], [0, 0, 1, 0], [0, 0, 0, 0], [9E9, 9E9, 9E9, 9E9, 9E9, 9E9]];
    CONST robtarget p14872:= [[1555.946649739784, -31.688077802945017, 1006.500033578516], [0, 0, 1, 0], [0, 0, 0, 0], [9E9, 9E9, 9E9, 9E9, 9E9, 9E9]];
    CONST robtarget p14873:= [[1555.6494613163316, -32.2091504840158, 1006.500033578516], [0, 0, 1, 0], [0, 0, 0, 0], [9E9, 9E9, 9E9, 9E9, 9E9, 9E9]];
    CONST robtarget p14874:= [[1555.230267057469, -32.89083445201545, 1006.500033578516], [0, 0, 1, 0], [0, 0, 0, 0], [9E9, 9E9, 9E9, 9E9, 9E9, 9E9]];
    CONST robtarget p14875:= [[1555.1759173813757, -32.997284302670195, 1006.500033578516], [0, 0, 1, 0], [0, 0, 0, 0], [9E9, 9E9, 9E9, 9E9, 9E9, 9E9]];
    CONST robtarget p14876:= [[1554.9004709995174, -33.437478603208845, 1006.500033578516], [0, 0, 1, 0], [0, 0, 0, 0], [9E9, 9E9, 9E9, 9E9, 9E9, 9E9]];
    CONST robtarget p14877:= [[1554.6762871984404, -33.81432530429322, 1006.500033578516], [0, 0, 1, 0], [0, 0, 0, 0], [9E9, 9E9, 9E9, 9E9, 9E9, 9E9]];
    CONST robtarget p14878:= [[1554.5705758733043, -33.99555072522356, 1006.500033578516], [0, 0, 1, 0], [0, 0, 0, 0], [9E9, 9E9, 9E9, 9E9, 9E9, 9E9]];
    CONST robtarget p14879:= [[1554.2451377823702, -34.532255855429646, 1006.500033578516], [0, 0, 1, 0], [0, 0, 0, 0], [9E9, 9E9, 9E9, 9E9, 9E9, 9E9]];
    CONST robtarget p14880:= [[1553.9908873674567, -34.949936863506345, 1006.500033578516], [0, 0, 1, 0], [0, 0, 0, 0], [9E9, 9E9, 9E9, 9E9, 9E9, 9E9]];
    CONST robtarget p14881:= [[1553.8138157226942, -35.217939548289664, 1006.500033578516], [0, 0, 1, 0], [0, 0, 0, 0], [9E9, 9E9, 9E9, 9E9, 9E9, 9E9]];
    CONST robtarget p14882:= [[1553.392911264964, -35.78661792551053, 1006.500033578516], [0, 0, 1, 0], [0, 0, 0, 0], [9E9, 9E9, 9E9, 9E9, 9E9, 9E9]];
    CONST robtarget p14883:= [[1552.862028420182, -36.580040499724184, 1006.500033578516], [0, 0, 1, 0], [0, 0, 0, 0], [9E9, 9E9, 9E9, 9E9, 9E9, 9E9]];
    CONST robtarget p14884:= [[1552.6604782340078, -36.88762681462611, 1006.500033578516], [0, 0, 1, 0], [0, 0, 0, 0], [9E9, 9E9, 9E9, 9E9, 9E9, 9E9]];
    CONST robtarget p14885:= [[1552.2868700574459, -37.38409220306884, 1006.500033578516], [0, 0, 1, 0], [0, 0, 0, 0], [9E9, 9E9, 9E9, 9E9, 9E9, 9E9]];
    CONST robtarget p14886:= [[1552.1146325569016, -37.6379196955306, 1006.500033578516], [0, 0, 1, 0], [0, 0, 0, 0], [9E9, 9E9, 9E9, 9E9, 9E9, 9E9]];
    CONST robtarget p14887:= [[1551.942310425491, -37.88913603015188, 1006.500033578516], [0, 0, 1, 0], [0, 0, 0, 0], [9E9, 9E9, 9E9, 9E9, 9E9, 9E9]];
    CONST robtarget p14888:= [[1551.3884675954043, -38.668899525244214, 1006.500033578516], [0, 0, 1, 0], [0, 0, 0, 0], [9E9, 9E9, 9E9, 9E9, 9E9, 9E9]];
    CONST robtarget p14889:= [[1551.0391311966882, -39.16639755431527, 1006.500033578516], [0, 0, 1, 0], [0, 0, 0, 0], [9E9, 9E9, 9E9, 9E9, 9E9, 9E9]];
    CONST robtarget p14890:= [[1550.5624850243612, -39.761288578653605, 1006.500033578516], [0, 0, 1, 0], [0, 0, 0, 0], [9E9, 9E9, 9E9, 9E9, 9E9, 9E9]];
    CONST robtarget p14891:= [[1550.1494975677442, -40.244883029476824, 1006.500033578516], [0, 0, 1, 0], [0, 0, 0, 0], [9E9, 9E9, 9E9, 9E9, 9E9, 9E9]];
    CONST robtarget p14892:= [[1549.507186059514, -40.98601492793843, 1006.500033578516], [0, 0, 1, 0], [0, 0, 0, 0], [9E9, 9E9, 9E9, 9E9, 9E9, 9E9]];
    CONST robtarget p14893:= [[1548.7842734850817, -41.80758116803424, 1006.500033578516], [0, 0, 1, 0], [0, 0, 0, 0], [9E9, 9E9, 9E9, 9E9, 9E9, 9E9]];
    CONST robtarget p14894:= [[1548.4048385161855, -42.28049077099923, 1006.500033578516], [0, 0, 1, 0], [0, 0, 0, 0], [9E9, 9E9, 9E9, 9E9, 9E9, 9E9]];
    CONST robtarget p14895:= [[1548.14685742254, -42.61495908614811, 1006.500033578516], [0, 0, 1, 0], [0, 0, 0, 0], [9E9, 9E9, 9E9, 9E9, 9E9, 9E9]];
    CONST robtarget p14896:= [[1547.8206643182662, -42.95346258235979, 1006.500033578516], [0, 0, 1, 0], [0, 0, 0, 0], [9E9, 9E9, 9E9, 9E9, 9E9, 9E9]];
    CONST robtarget p14897:= [[1547.3768306164466, -43.48345004581816, 1006.500033578516], [0, 0, 1, 0], [0, 0, 0, 0], [9E9, 9E9, 9E9, 9E9, 9E9, 9E9]];
    CONST robtarget p14898:= [[1547.157129292676, -43.714600676272696, 1006.500033578516], [0, 0, 1, 0], [0, 0, 0, 0], [9E9, 9E9, 9E9, 9E9, 9E9, 9E9]];
    CONST robtarget p14899:= [[1546.7355201795142, -44.143505692122034, 1006.500033578516], [0, 0, 1, 0], [0, 0, 0, 0], [9E9, 9E9, 9E9, 9E9, 9E9, 9E9]];
    CONST robtarget p14900:= [[1546.2346450296059, -44.66430636079644, 1006.500033578516], [0, 0, 1, 0], [0, 0, 0, 0], [9E9, 9E9, 9E9, 9E9, 9E9, 9E9]];
    CONST robtarget p14901:= [[1545.729149716231, -45.139964448899846, 1006.500033578516], [0, 0, 1, 0], [0, 0, 0, 0], [9E9, 9E9, 9E9, 9E9, 9E9, 9E9]];
    CONST robtarget p14902:= [[1545.4546858696367, -45.40338824852229, 1006.500033578516], [0, 0, 1, 0], [0, 0, 0, 0], [9E9, 9E9, 9E9, 9E9, 9E9, 9E9]];
    CONST robtarget p14903:= [[1544.744626316363, -46.213366046542234, 1006.500033578516], [0, 0, 1, 0], [0, 0, 0, 0], [9E9, 9E9, 9E9, 9E9, 9E9, 9E9]];
    CONST robtarget p14904:= [[1544.6892413004332, -46.280300469696485, 1006.500033578516], [0, 0, 1, 0], [0, 0, 0, 0], [9E9, 9E9, 9E9, 9E9, 9E9, 9E9]];
    CONST robtarget p14905:= [[1544.3398068760976, -46.602831586353616, 1006.500033578516], [0, 0, 1, 0], [0, 0, 0, 0], [9E9, 9E9, 9E9, 9E9, 9E9, 9E9]];
    CONST robtarget p14906:= [[1544.0339529102373, -46.86481374873988, 1006.500033578516], [0, 0, 1, 0], [0, 0, 0, 0], [9E9, 9E9, 9E9, 9E9, 9E9, 9E9]];
    CONST robtarget p14907:= [[1543.9048347841313, -46.983331662336305, 1006.500033578516], [0, 0, 1, 0], [0, 0, 0, 0], [9E9, 9E9, 9E9, 9E9, 9E9, 9E9]];
    CONST robtarget p14908:= [[1543.5507309412026, -47.31060360838974, 1006.500033578516], [0, 0, 1, 0], [0, 0, 0, 0], [9E9, 9E9, 9E9, 9E9, 9E9, 9E9]];
    CONST robtarget p14909:= [[1542.8174608205597, -47.91797906627021, 1006.500033578516], [0, 0, 1, 0], [0, 0, 0, 0], [9E9, 9E9, 9E9, 9E9, 9E9, 9E9]];
    CONST robtarget p14910:= [[1542.57824113613, -48.167417421675125, 1006.500033578516], [0, 0, 1, 0], [0, 0, 0, 0], [9E9, 9E9, 9E9, 9E9, 9E9, 9E9]];
    CONST robtarget p14911:= [[1542.5247769376288, -48.2236738567885, 1006.500033578516], [0, 0, 1, 0], [0, 0, 0, 0], [9E9, 9E9, 9E9, 9E9, 9E9, 9E9]];
    CONST robtarget p14912:= [[1542.0710921951568, -48.60859780896561, 1006.500033578516], [0, 0, 1, 0], [0, 0, 0, 0], [9E9, 9E9, 9E9, 9E9, 9E9, 9E9]];
    CONST robtarget p14913:= [[1541.796272663009, -48.84136738551912, 1006.500033578516], [0, 0, 1, 0], [0, 0, 0, 0], [9E9, 9E9, 9E9, 9E9, 9E9, 9E9]];
    CONST robtarget p14914:= [[1541.4377706744383, -49.15576841129092, 1006.500033578516], [0, 0, 1, 0], [0, 0, 0, 0], [9E9, 9E9, 9E9, 9E9, 9E9, 9E9]];
    CONST robtarget p14915:= [[1541.1380021805737, -49.45808925904888, 1006.500033578516], [0, 0, 1, 0], [0, 0, 0, 0], [9E9, 9E9, 9E9, 9E9, 9E9, 9E9]];
    CONST robtarget p14916:= [[1540.6680421912522, -49.801037846109665, 1006.500033578516], [0, 0, 1, 0], [0, 0, 0, 0], [9E9, 9E9, 9E9, 9E9, 9E9, 9E9]];
    CONST robtarget p14917:= [[1540.46407384905, -49.97805268059918, 1006.500033578516], [0, 0, 1, 0], [0, 0, 0, 0], [9E9, 9E9, 9E9, 9E9, 9E9, 9E9]];
    CONST robtarget p14918:= [[1539.8670838620096, -50.444724874197064, 1006.500033578516], [0, 0, 1, 0], [0, 0, 0, 0], [9E9, 9E9, 9E9, 9E9, 9E9, 9E9]];
    CONST robtarget p14919:= [[1539.599394978819, -50.6555901745958, 1006.500033578516], [0, 0, 1, 0], [0, 0, 0, 0], [9E9, 9E9, 9E9, 9E9, 9E9, 9E9]];
    CONST robtarget p14920:= [[1538.4730722184472, -51.468405788805526, 1006.500033578516], [0, 0, 1, 0], [0, 0, 0, 0], [9E9, 9E9, 9E9, 9E9, 9E9, 9E9]];
    CONST robtarget p14921:= [[1538.3763776649098, -51.554924320903496, 1006.500033578516], [0, 0, 1, 0], [0, 0, 0, 0], [9E9, 9E9, 9E9, 9E9, 9E9, 9E9]];
    CONST robtarget p14922:= [[1537.7603133023654, -52.053850191111636, 1006.500033578516], [0, 0, 1, 0], [0, 0, 0, 0], [9E9, 9E9, 9E9, 9E9, 9E9, 9E9]];
    CONST robtarget p14923:= [[1537.6646286080588, -52.14651426079008, 1006.500033578516], [0, 0, 1, 0], [0, 0, 0, 0], [9E9, 9E9, 9E9, 9E9, 9E9, 9E9]];
    CONST robtarget p14924:= [[1537.3840678782974, -52.34853087345344, 1006.500033578516], [0, 0, 1, 0], [0, 0, 0, 0], [9E9, 9E9, 9E9, 9E9, 9E9, 9E9]];
    CONST robtarget p14925:= [[1536.818363877833, -52.690751751305406, 1006.500033578516], [0, 0, 1, 0], [0, 0, 0, 0], [9E9, 9E9, 9E9, 9E9, 9E9, 9E9]];
    CONST robtarget p14926:= [[1536.3769787024721, -52.98187604510281, 1006.500033578516], [0, 0, 1, 0], [0, 0, 0, 0], [9E9, 9E9, 9E9, 9E9, 9E9, 9E9]];
    CONST robtarget p14927:= [[1536.1647391975264, -53.14483639020042, 1006.500033578516], [0, 0, 1, 0], [0, 0, 0, 0], [9E9, 9E9, 9E9, 9E9, 9E9, 9E9]];
    CONST robtarget p14928:= [[1535.758144836897, -53.43067996792179, 1006.500033578516], [0, 0, 1, 0], [0, 0, 0, 0], [9E9, 9E9, 9E9, 9E9, 9E9, 9E9]];
    CONST robtarget p14929:= [[1535.2460057956982, -53.76954292415113, 1006.500033578516], [0, 0, 1, 0], [0, 0, 0, 0], [9E9, 9E9, 9E9, 9E9, 9E9, 9E9]];
    CONST robtarget p14930:= [[1534.7302086549578, -54.09554400564303, 1006.500033578516], [0, 0, 1, 0], [0, 0, 0, 0], [9E9, 9E9, 9E9, 9E9, 9E9, 9E9]];
    CONST robtarget p14931:= [[1534.1608480575608, -54.476166954899476, 1006.500033578516], [0, 0, 1, 0], [0, 0, 0, 0], [9E9, 9E9, 9E9, 9E9, 9E9, 9E9]];
    CONST robtarget p14932:= [[1533.9180539039144, -54.64953275855822, 1006.500033578516], [0, 0, 1, 0], [0, 0, 0, 0], [9E9, 9E9, 9E9, 9E9, 9E9, 9E9]];
    CONST robtarget p14933:= [[1533.179355411489, -55.081532081542505, 1006.500033578516], [0, 0, 1, 0], [0, 0, 0, 0], [9E9, 9E9, 9E9, 9E9, 9E9, 9E9]];
    CONST robtarget p14934:= [[1532.8052589631072, -55.32326989394186, 1006.500033578516], [0, 0, 1, 0], [0, 0, 0, 0], [9E9, 9E9, 9E9, 9E9, 9E9, 9E9]];
    CONST robtarget p14935:= [[1531.9485129768952, -55.802641917513235, 1006.500033578516], [0, 0, 1, 0], [0, 0, 0, 0], [9E9, 9E9, 9E9, 9E9, 9E9, 9E9]];
    CONST robtarget p14936:= [[1531.4107754306285, -56.1032246113668, 1006.500033578516], [0, 0, 1, 0], [0, 0, 0, 0], [9E9, 9E9, 9E9, 9E9, 9E9, 9E9]];
    CONST robtarget p14937:= [[1530.8405016701597, -56.42474356157126, 1006.500033578516], [0, 0, 1, 0], [0, 0, 0, 0], [9E9, 9E9, 9E9, 9E9, 9E9, 9E9]];
    CONST robtarget p14938:= [[1530.1452460148066, -56.778752769448865, 1006.500033578516], [0, 0, 1, 0], [0, 0, 0, 0], [9E9, 9E9, 9E9, 9E9, 9E9, 9E9]];
    CONST robtarget p14939:= [[1529.88242518332, -56.9390323195773, 1006.500033578516], [0, 0, 1, 0], [0, 0, 0, 0], [9E9, 9E9, 9E9, 9E9, 9E9, 9E9]];
    CONST robtarget p14940:= [[1529.5396122432858, -57.15324342244994, 1006.500033578516], [0, 0, 1, 0], [0, 0, 0, 0], [9E9, 9E9, 9E9, 9E9, 9E9, 9E9]];
    CONST robtarget p14941:= [[1529.1999792447114, -57.316170931035245, 1006.500033578516], [0, 0, 1, 0], [0, 0, 0, 0], [9E9, 9E9, 9E9, 9E9, 9E9, 9E9]];
    CONST robtarget p14942:= [[1529.1332090141698, -57.34717481010436, 1006.500033578516], [0, 0, 1, 0], [0, 0, 0, 0], [9E9, 9E9, 9E9, 9E9, 9E9, 9E9]];
    CONST robtarget p14943:= [[1528.6060366793597, -57.59444895759974, 1006.500033578516], [0, 0, 1, 0], [0, 0, 0, 0], [9E9, 9E9, 9E9, 9E9, 9E9, 9E9]];
    CONST robtarget p14944:= [[1527.702291783923, -58.02803791531328, 1006.500033578516], [0, 0, 1, 0], [0, 0, 0, 0], [9E9, 9E9, 9E9, 9E9, 9E9, 9E9]];
    CONST robtarget p14945:= [[1527.4248322371118, -58.12764542675508, 1006.500033578516], [0, 0, 1, 0], [0, 0, 0, 0], [9E9, 9E9, 9E9, 9E9, 9E9, 9E9]];
    CONST robtarget p14946:= [[1526.605321622362, -58.53968958126637, 1006.500033578516], [0, 0, 1, 0], [0, 0, 0, 0], [9E9, 9E9, 9E9, 9E9, 9E9, 9E9]];
    CONST robtarget p14947:= [[1526.1902669128035, -58.7341195399214, 1006.500033578516], [0, 0, 1, 0], [0, 0, 0, 0], [9E9, 9E9, 9E9, 9E9, 9E9, 9E9]];
    CONST robtarget p14948:= [[1525.789614795063, -58.914125864760734, 1006.500033578516], [0, 0, 1, 0], [0, 0, 0, 0], [9E9, 9E9, 9E9, 9E9, 9E9, 9E9]];
    CONST robtarget p14949:= [[1525.0014209815508, -59.23879887230835, 1006.500033578516], [0, 0, 1, 0], [0, 0, 0, 0], [9E9, 9E9, 9E9, 9E9, 9E9, 9E9]];
    CONST robtarget p14950:= [[1524.1973952821418, -59.5743085968531, 1006.500033578516], [0, 0, 1, 0], [0, 0, 0, 0], [9E9, 9E9, 9E9, 9E9, 9E9, 9E9]];
    CONST robtarget p14951:= [[1523.9634539823503, -59.67640164867346, 1006.500033578516], [0, 0, 1, 0], [0, 0, 0, 0], [9E9, 9E9, 9E9, 9E9, 9E9, 9E9]];
    CONST robtarget p14952:= [[1523.417669620706, -59.876091808734195, 1006.500033578516], [0, 0, 1, 0], [0, 0, 0, 0], [9E9, 9E9, 9E9, 9E9, 9E9, 9E9]];
    CONST robtarget p14953:= [[1523.3267745164987, -59.915053859794085, 1006.500033578516], [0, 0, 1, 0], [0, 0, 0, 0], [9E9, 9E9, 9E9, 9E9, 9E9, 9E9]];
    CONST robtarget p14954:= [[1522.303843566067, -60.302971663857136, 1006.500033578516], [0, 0, 1, 0], [0, 0, 0, 0], [9E9, 9E9, 9E9, 9E9, 9E9, 9E9]];
    CONST robtarget p14955:= [[1521.7708636110103, -60.50855689319797, 1006.500033578516], [0, 0, 1, 0], [0, 0, 0, 0], [9E9, 9E9, 9E9, 9E9, 9E9, 9E9]];
    CONST robtarget p14956:= [[1521.3329471861955, -60.66575026111912, 1006.500033578516], [0, 0, 1, 0], [0, 0, 0, 0], [9E9, 9E9, 9E9, 9E9, 9E9, 9E9]];
    CONST robtarget p14957:= [[1521.2022029386544, -60.714984859665535, 1006.500033578516], [0, 0, 1, 0], [0, 0, 0, 0], [9E9, 9E9, 9E9, 9E9, 9E9, 9E9]];
    CONST robtarget p14958:= [[1520.5697203869322, -60.958289538265134, 1006.500033578516], [0, 0, 1, 0], [0, 0, 0, 0], [9E9, 9E9, 9E9, 9E9, 9E9, 9E9]];
    CONST robtarget p14959:= [[1520.3191326502217, -61.021541254814544, 1006.500033578516], [0, 0, 1, 0], [0, 0, 0, 0], [9E9, 9E9, 9E9, 9E9, 9E9, 9E9]];
    CONST robtarget p14960:= [[1519.166329863163, -61.37811312878308, 1006.500033578516], [0, 0, 1, 0], [0, 0, 0, 0], [9E9, 9E9, 9E9, 9E9, 9E9, 9E9]];
    CONST robtarget p14961:= [[1518.5370970443669, -61.557239285961344, 1006.500033578516], [0, 0, 1, 0], [0, 0, 0, 0], [9E9, 9E9, 9E9, 9E9, 9E9, 9E9]];
    CONST robtarget p14962:= [[1518.3278128932543, -61.62891548850246, 1006.500033578516], [0, 0, 1, 0], [0, 0, 0, 0], [9E9, 9E9, 9E9, 9E9, 9E9, 9E9]];
    CONST robtarget p14963:= [[1517.9740704709877, -61.72345365572395, 1006.500033578516], [0, 0, 1, 0], [0, 0, 0, 0], [9E9, 9E9, 9E9, 9E9, 9E9, 9E9]];
    CONST robtarget p14964:= [[1517.3447793829673, -61.88487261741833, 1006.500033578516], [0, 0, 1, 0], [0, 0, 0, 0], [9E9, 9E9, 9E9, 9E9, 9E9, 9E9]];
    CONST robtarget p14965:= [[1516.8365585274967, -62.07871820893638, 1006.500033578516], [0, 0, 1, 0], [0, 0, 0, 0], [9E9, 9E9, 9E9, 9E9, 9E9, 9E9]];
    CONST robtarget p14966:= [[1516.2235660550996, -62.23907140379965, 1006.500033578516], [0, 0, 1, 0], [0, 0, 0, 0], [9E9, 9E9, 9E9, 9E9, 9E9, 9E9]];
    CONST robtarget p14967:= [[1515.6234014734891, -62.39547595040773, 1006.500033578516], [0, 0, 1, 0], [0, 0, 0, 0], [9E9, 9E9, 9E9, 9E9, 9E9, 9E9]];
    CONST robtarget p14968:= [[1514.4848193464259, -62.631255722264314, 1006.500033578516], [0, 0, 1, 0], [0, 0, 0, 0], [9E9, 9E9, 9E9, 9E9, 9E9, 9E9]];
    CONST robtarget p14969:= [[1514.3383903862941, -62.67670004245866, 1006.500033578516], [0, 0, 1, 0], [0, 0, 0, 0], [9E9, 9E9, 9E9, 9E9, 9E9, 9E9]];
    CONST robtarget p14970:= [[1514.0529603198731, -62.724991761052564, 1006.500033578516], [0, 0, 1, 0], [0, 0, 0, 0], [9E9, 9E9, 9E9, 9E9, 9E9, 9E9]];
    CONST robtarget p14971:= [[1513.2365660131602, -62.871757706385274, 1006.500033578516], [0, 0, 1, 0], [0, 0, 0, 0], [9E9, 9E9, 9E9, 9E9, 9E9, 9E9]];
    CONST robtarget p14972:= [[1512.7130421308027, -63.015574595969554, 1006.500033578516], [0, 0, 1, 0], [0, 0, 0, 0], [9E9, 9E9, 9E9, 9E9, 9E9, 9E9]];
    CONST robtarget p14973:= [[1512.4365089802377, -63.105660811770406, 1006.500033578516], [0, 0, 1, 0], [0, 0, 0, 0], [9E9, 9E9, 9E9, 9E9, 9E9, 9E9]];
    CONST robtarget p14974:= [[1512.2670833465118, -63.13526943133706, 1006.500033578516], [0, 0, 1, 0], [0, 0, 0, 0], [9E9, 9E9, 9E9, 9E9, 9E9, 9E9]];
    CONST robtarget p14975:= [[1511.6391558870935, -63.27968465532297, 1006.500033578516], [0, 0, 1, 0], [0, 0, 0, 0], [9E9, 9E9, 9E9, 9E9, 9E9, 9E9]];
    CONST robtarget p14976:= [[1511.399694023771, -63.30998073977109, 1006.500033578516], [0, 0, 1, 0], [0, 0, 0, 0], [9E9, 9E9, 9E9, 9E9, 9E9, 9E9]];
    CONST robtarget p14977:= [[1510.90867658619, -63.373986252916154, 1006.500033578516], [0, 0, 1, 0], [0, 0, 0, 0], [9E9, 9E9, 9E9, 9E9, 9E9, 9E9]];
    CONST robtarget p14978:= [[1510.7269588103657, -63.40738118411778, 1006.500033578516], [0, 0, 1, 0], [0, 0, 0, 0], [9E9, 9E9, 9E9, 9E9, 9E9, 9E9]];
    CONST robtarget p14979:= [[1510.0380796991103, -63.50127482494363, 1006.500033578516], [0, 0, 1, 0], [0, 0, 0, 0], [9E9, 9E9, 9E9, 9E9, 9E9, 9E9]];
    CONST robtarget p14980:= [[1509.8182834396766, -63.53854123476616, 1006.500033578516], [0, 0, 1, 0], [0, 0, 0, 0], [9E9, 9E9, 9E9, 9E9, 9E9, 9E9]];
    CONST robtarget p14981:= [[1509.2605001991235, -63.62017249381609, 1006.500033578516], [0, 0, 1, 0], [0, 0, 0, 0], [9E9, 9E9, 9E9, 9E9, 9E9, 9E9]];
    CONST robtarget p14982:= [[1508.768839978461, -63.69378284135223, 1006.500033578516], [0, 0, 1, 0], [0, 0, 0, 0], [9E9, 9E9, 9E9, 9E9, 9E9, 9E9]];
    CONST robtarget p14983:= [[1508.0477337183293, -63.775905848138834, 1006.500033578516], [0, 0, 1, 0], [0, 0, 0, 0], [9E9, 9E9, 9E9, 9E9, 9E9, 9E9]];
    CONST robtarget p14984:= [[1507.7825741593392, -63.8266263701248, 1006.500033578516], [0, 0, 1, 0], [0, 0, 0, 0], [9E9, 9E9, 9E9, 9E9, 9E9, 9E9]];
    CONST robtarget p14985:= [[1507.263898917035, -63.92328816541193, 1006.500033578516], [0, 0, 1, 0], [0, 0, 0, 0], [9E9, 9E9, 9E9, 9E9, 9E9, 9E9]];
    CONST robtarget p14986:= [[1506.745439227206, -63.96569050759804, 1006.500033578516], [0, 0, 1, 0], [0, 0, 0, 0], [9E9, 9E9, 9E9, 9E9, 9E9, 9E9]];
    CONST robtarget p14987:= [[1505.7862877238908, -64.01036569741386, 1006.500033578516], [0, 0, 1, 0], [0, 0, 0, 0], [9E9, 9E9, 9E9, 9E9, 9E9, 9E9]];
    CONST robtarget p14988:= [[1505.1924623102002, -64.06974900485413, 1006.500033578516], [0, 0, 1, 0], [0, 0, 0, 0], [9E9, 9E9, 9E9, 9E9, 9E9, 9E9]];
    CONST robtarget p14989:= [[1504.757346550164, -64.11856732887581, 1006.500033578516], [0, 0, 1, 0], [0, 0, 0, 0], [9E9, 9E9, 9E9, 9E9, 9E9, 9E9]];
    CONST robtarget p14990:= [[1504.4344805969386, -64.1412560982914, 1006.500033578516], [0, 0, 1, 0], [0, 0, 0, 0], [9E9, 9E9, 9E9, 9E9, 9E9, 9E9]];
    CONST robtarget p14991:= [[1503.9947809117898, -64.14855405570937, 1006.500033578516], [0, 0, 1, 0], [0, 0, 0, 0], [9E9, 9E9, 9E9, 9E9, 9E9, 9E9]];
    CONST robtarget p14992:= [[1503.0036785747964, -64.24898935397432, 1006.500033578516], [0, 0, 1, 0], [0, 0, 0, 0], [9E9, 9E9, 9E9, 9E9, 9E9, 9E9]];
    CONST robtarget p14993:= [[1502.4659019425603, -64.29145085468991, 1006.500033578516], [0, 0, 1, 0], [0, 0, 0, 0], [9E9, 9E9, 9E9, 9E9, 9E9, 9E9]];
    CONST robtarget p14994:= [[1502.208042500626, -64.30325536587111, 1006.500033578516], [0, 0, 1, 0], [0, 0, 0, 0], [9E9, 9E9, 9E9, 9E9, 9E9, 9E9]];
    CONST robtarget p14995:= [[1501.7168399234804, -64.29494755224326, 1006.500033578516], [0, 0, 1, 0], [0, 0, 0, 0], [9E9, 9E9, 9E9, 9E9, 9E9, 9E9]];
    CONST robtarget p14996:= [[1501.0464139424316, -64.27980960111057, 1006.500033578516], [0, 0, 1, 0], [0, 0, 0, 0], [9E9, 9E9, 9E9, 9E9, 9E9, 9E9]];
    CONST robtarget p14997:= [[1500.5876677209349, -64.29577576369324, 1006.500033578516], [0, 0, 1, 0], [0, 0, 0, 0], [9E9, 9E9, 9E9, 9E9, 9E9, 9E9]];
    CONST robtarget p14998:= [[1500.333384165863, -64.29108833959631, 1006.500033578516], [0, 0, 1, 0], [0, 0, 0, 0], [9E9, 9E9, 9E9, 9E9, 9E9, 9E9]];
    CONST robtarget p14999:= [[1499.2457669483515, -64.29711659222467, 1006.500033578516], [0, 0, 1, 0], [0, 0, 0, 0], [9E9, 9E9, 9E9, 9E9, 9E9, 9E9]];
    CONST robtarget p15000:= [[1498.322267942967, -64.26530634023524, 1006.500033578516], [0, 0, 1, 0], [0, 0, 0, 0], [9E9, 9E9, 9E9, 9E9, 9E9, 9E9]];
    CONST robtarget p15001:= [[1497.692916975533, -64.2474835361183, 1006.500033578516], [0, 0, 1, 0], [0, 0, 0, 0], [9E9, 9E9, 9E9, 9E9, 9E9, 9E9]];
    CONST robtarget p15002:= [[1497.2594456741156, -64.26902766415003, 1006.500033578516], [0, 0, 1, 0], [0, 0, 0, 0], [9E9, 9E9, 9E9, 9E9, 9E9, 9E9]];
    CONST robtarget p15003:= [[1496.96664801538, -64.24259888921925, 1006.500033578516], [0, 0, 1, 0], [0, 0, 0, 0], [9E9, 9E9, 9E9, 9E9, 9E9, 9E9]];
    CONST robtarget p15004:= [[1496.1934421391759, -64.19632708835275, 1006.500033578516], [0, 0, 1, 0], [0, 0, 0, 0], [9E9, 9E9, 9E9, 9E9, 9E9, 9E9]];
    CONST robtarget p15005:= [[1495.7306293696458, -64.12547734049377, 1006.500033578516], [0, 0, 1, 0], [0, 0, 0, 0], [9E9, 9E9, 9E9, 9E9, 9E9, 9E9]];
    CONST robtarget p15006:= [[1495.1244216261107, -64.08731100511163, 1006.500033578516], [0, 0, 1, 0], [0, 0, 0, 0], [9E9, 9E9, 9E9, 9E9, 9E9, 9E9]];
    CONST robtarget p15007:= [[1494.658606825372, -64.06192400214233, 1006.500033578516], [0, 0, 1, 0], [0, 0, 0, 0], [9E9, 9E9, 9E9, 9E9, 9E9, 9E9]];
    CONST robtarget p15008:= [[1494.349738180898, -64.06221985397784, 1006.500033578516], [0, 0, 1, 0], [0, 0, 0, 0], [9E9, 9E9, 9E9, 9E9, 9E9, 9E9]];
    CONST robtarget p15009:= [[1493.485595983013, -63.97813389956004, 1006.500033578516], [0, 0, 1, 0], [0, 0, 0, 0], [9E9, 9E9, 9E9, 9E9, 9E9, 9E9]];
    CONST robtarget p15010:= [[1493.0383064742598, -63.96430811144376, 1006.500033578516], [0, 0, 1, 0], [0, 0, 0, 0], [9E9, 9E9, 9E9, 9E9, 9E9, 9E9]];
    CONST robtarget p15011:= [[1492.8239968626906, -63.9361093653834, 1006.500033578516], [0, 0, 1, 0], [0, 0, 0, 0], [9E9, 9E9, 9E9, 9E9, 9E9, 9E9]];
    CONST robtarget p15012:= [[1491.9737862352038, -63.813702619652325, 1006.500033578516], [0, 0, 1, 0], [0, 0, 0, 0], [9E9, 9E9, 9E9, 9E9, 9E9, 9E9]];
    CONST robtarget p15013:= [[1491.8183091413464, -63.77170703723101, 1006.500033578516], [0, 0, 1, 0], [0, 0, 0, 0], [9E9, 9E9, 9E9, 9E9, 9E9, 9E9]];
    CONST robtarget p15014:= [[1490.6012743476342, -63.56664554322278, 1006.500033578516], [0, 0, 1, 0], [0, 0, 0, 0], [9E9, 9E9, 9E9, 9E9, 9E9, 9E9]];
    CONST robtarget p15015:= [[1490.2043212645528, -63.510361429143195, 1006.500033578516], [0, 0, 1, 0], [0, 0, 0, 0], [9E9, 9E9, 9E9, 9E9, 9E9, 9E9]];
    CONST robtarget p15016:= [[1489.796767742938, -63.47899299079757, 1006.500033578516], [0, 0, 1, 0], [0, 0, 0, 0], [9E9, 9E9, 9E9, 9E9, 9E9, 9E9]];
    CONST robtarget p15017:= [[1489.4712199677085, -63.44075805307611, 1006.500033578516], [0, 0, 1, 0], [0, 0, 0, 0], [9E9, 9E9, 9E9, 9E9, 9E9, 9E9]];
    CONST robtarget p15018:= [[1489.2243503117502, -63.41052387217047, 1006.500033578516], [0, 0, 1, 0], [0, 0, 0, 0], [9E9, 9E9, 9E9, 9E9, 9E9, 9E9]];
    CONST robtarget p15019:= [[1488.8065500986436, -63.327006840926565, 1006.500033578516], [0, 0, 1, 0], [0, 0, 0, 0], [9E9, 9E9, 9E9, 9E9, 9E9, 9E9]];
    CONST robtarget p15020:= [[1488.1975747964652, -63.23548203900089, 1006.500033578516], [0, 0, 1, 0], [0, 0, 0, 0], [9E9, 9E9, 9E9, 9E9, 9E9, 9E9]];
    CONST robtarget p15021:= [[1487.6410525391725, -63.086056304931034, 1006.500033578516], [0, 0, 1, 0], [0, 0, 0, 0], [9E9, 9E9, 9E9, 9E9, 9E9, 9E9]];
    CONST robtarget p15022:= [[1487.393988287071, -63.0168889969168, 1006.500033578516], [0, 0, 1, 0], [0, 0, 0, 0], [9E9, 9E9, 9E9, 9E9, 9E9, 9E9]];
    CONST robtarget p15023:= [[1486.2466992640043, -62.79345904730255, 1006.500033578516], [0, 0, 1, 0], [0, 0, 0, 0], [9E9, 9E9, 9E9, 9E9, 9E9, 9E9]];
    CONST robtarget p15024:= [[1485.5098658007987, -62.640630572352386, 1006.500033578516], [0, 0, 1, 0], [0, 0, 0, 0], [9E9, 9E9, 9E9, 9E9, 9E9, 9E9]];
    CONST robtarget p15025:= [[1485.262644636248, -62.59473202517603, 1006.500033578516], [0, 0, 1, 0], [0, 0, 0, 0], [9E9, 9E9, 9E9, 9E9, 9E9, 9E9]];
    CONST robtarget p15026:= [[1484.7440536895651, -62.4762393500964, 1006.500033578516], [0, 0, 1, 0], [0, 0, 0, 0], [9E9, 9E9, 9E9, 9E9, 9E9, 9E9]];
    CONST robtarget p15027:= [[1484.5911910978025, -62.43986211171968, 1006.500033578516], [0, 0, 1, 0], [0, 0, 0, 0], [9E9, 9E9, 9E9, 9E9, 9E9, 9E9]];
    CONST robtarget p15028:= [[1484.4344122903613, -62.38791037773487, 1006.500033578516], [0, 0, 1, 0], [0, 0, 0, 0], [9E9, 9E9, 9E9, 9E9, 9E9, 9E9]];
    CONST robtarget p15029:= [[1483.7376184725802, -62.22277032072221, 1006.500033578516], [0, 0, 1, 0], [0, 0, 0, 0], [9E9, 9E9, 9E9, 9E9, 9E9, 9E9]];
    CONST robtarget p15030:= [[1483.2917963122495, -62.1141306213667, 1006.500033578516], [0, 0, 1, 0], [0, 0, 0, 0], [9E9, 9E9, 9E9, 9E9, 9E9, 9E9]];
    CONST robtarget p15031:= [[1482.9367183780735, -61.99305391381701, 1006.500033578516], [0, 0, 1, 0], [0, 0, 0, 0], [9E9, 9E9, 9E9, 9E9, 9E9, 9E9]];
    CONST robtarget p15032:= [[1482.5315323075151, -61.880384237199884, 1006.500033578516], [0, 0, 1, 0], [0, 0, 0, 0], [9E9, 9E9, 9E9, 9E9, 9E9, 9E9]];
    CONST robtarget p15033:= [[1481.6709338049873, -61.6173119703136, 1006.500033578516], [0, 0, 1, 0], [0, 0, 0, 0], [9E9, 9E9, 9E9, 9E9, 9E9, 9E9]];
    CONST robtarget p15034:= [[1481.382083656706, -61.54225459603125, 1006.500033578516], [0, 0, 1, 0], [0, 0, 0, 0], [9E9, 9E9, 9E9, 9E9, 9E9, 9E9]];
    CONST robtarget p15035:= [[1480.951817209814, -61.41945581603823, 1006.500033578516], [0, 0, 1, 0], [0, 0, 0, 0], [9E9, 9E9, 9E9, 9E9, 9E9, 9E9]];
    CONST robtarget p15036:= [[1480.7431862188328, -61.340052594219394, 1006.500033578516], [0, 0, 1, 0], [0, 0, 0, 0], [9E9, 9E9, 9E9, 9E9, 9E9, 9E9]];
    CONST robtarget p15037:= [[1479.864223120338, -61.08809720815387, 1006.500033578516], [0, 0, 1, 0], [0, 0, 0, 0], [9E9, 9E9, 9E9, 9E9, 9E9, 9E9]];
    CONST robtarget p15038:= [[1479.6357568783123, -61.017963476209765, 1006.500033578516], [0, 0, 1, 0], [0, 0, 0, 0], [9E9, 9E9, 9E9, 9E9, 9E9, 9E9]];
    CONST robtarget p15039:= [[1479.5726732830876, -60.98852567251582, 1006.500033578516], [0, 0, 1, 0], [0, 0, 0, 0], [9E9, 9E9, 9E9, 9E9, 9E9, 9E9]];
    CONST robtarget p15040:= [[1478.9270321397594, -60.73013403431542, 1006.500033578516], [0, 0, 1, 0], [0, 0, 0, 0], [9E9, 9E9, 9E9, 9E9, 9E9, 9E9]];
    CONST robtarget p15041:= [[1478.4278450045406, -60.57611737429764, 1006.500033578516], [0, 0, 1, 0], [0, 0, 0, 0], [9E9, 9E9, 9E9, 9E9, 9E9, 9E9]];
    CONST robtarget p15042:= [[1477.5231505814356, -60.248334645012164, 1006.500033578516], [0, 0, 1, 0], [0, 0, 0, 0], [9E9, 9E9, 9E9, 9E9, 9E9, 9E9]];
    CONST robtarget p15043:= [[1477.2338708426826, -60.13469464019399, 1006.500033578516], [0, 0, 1, 0], [0, 0, 0, 0], [9E9, 9E9, 9E9, 9E9, 9E9, 9E9]];
    CONST robtarget p15044:= [[1476.6793480468536, -59.927877964619995, 1006.500033578516], [0, 0, 1, 0], [0, 0, 0, 0], [9E9, 9E9, 9E9, 9E9, 9E9, 9E9]];
    CONST robtarget p15045:= [[1476.6174675577097, -59.90152962372295, 1006.500033578516], [0, 0, 1, 0], [0, 0, 0, 0], [9E9, 9E9, 9E9, 9E9, 9E9, 9E9]];
    CONST robtarget p15046:= [[1476.149856769257, -59.69606943258527, 1006.500033578516], [0, 0, 1, 0], [0, 0, 0, 0], [9E9, 9E9, 9E9, 9E9, 9E9, 9E9]];
    CONST robtarget p15047:= [[1475.193060641743, -59.350486530811374, 1006.500033578516], [0, 0, 1, 0], [0, 0, 0, 0], [9E9, 9E9, 9E9, 9E9, 9E9, 9E9]];
    CONST robtarget p15048:= [[1474.8777945936365, -59.22799575282656, 1006.500033578516], [0, 0, 1, 0], [0, 0, 0, 0], [9E9, 9E9, 9E9, 9E9, 9E9, 9E9]];
    CONST robtarget p15049:= [[1474.4651837466672, -59.01967225379241, 1006.500033578516], [0, 0, 1, 0], [0, 0, 0, 0], [9E9, 9E9, 9E9, 9E9, 9E9, 9E9]];
    CONST robtarget p15050:= [[1473.7188040509195, -58.66605837616638, 1006.500033578516], [0, 0, 1, 0], [0, 0, 0, 0], [9E9, 9E9, 9E9, 9E9, 9E9, 9E9]];
    CONST robtarget p15051:= [[1473.3776092941312, -58.52821508597306, 1006.500033578516], [0, 0, 1, 0], [0, 0, 0, 0], [9E9, 9E9, 9E9, 9E9, 9E9, 9E9]];
    CONST robtarget p15052:= [[1472.7566566578987, -58.222733256506814, 1006.500033578516], [0, 0, 1, 0], [0, 0, 0, 0], [9E9, 9E9, 9E9, 9E9, 9E9, 9E9]];
    CONST robtarget p15053:= [[1472.4321585370283, -58.096772959423554, 1006.500033578516], [0, 0, 1, 0], [0, 0, 0, 0], [9E9, 9E9, 9E9, 9E9, 9E9, 9E9]];
    CONST robtarget p15054:= [[1471.1242293126243, -57.47562018219702, 1006.500033578516], [0, 0, 1, 0], [0, 0, 0, 0], [9E9, 9E9, 9E9, 9E9, 9E9, 9E9]];
    CONST robtarget p15055:= [[1470.819827222745, -57.30749896919037, 1006.500033578516], [0, 0, 1, 0], [0, 0, 0, 0], [9E9, 9E9, 9E9, 9E9, 9E9, 9E9]];
    CONST robtarget p15056:= [[1470.3279643502415, -57.07507503559381, 1006.500033578516], [0, 0, 1, 0], [0, 0, 0, 0], [9E9, 9E9, 9E9, 9E9, 9E9, 9E9]];
    CONST robtarget p15057:= [[1470.2278823484103, -57.02057987369162, 1006.500033578516], [0, 0, 1, 0], [0, 0, 0, 0], [9E9, 9E9, 9E9, 9E9, 9E9, 9E9]];
    CONST robtarget p15058:= [[1469.2780437226847, -56.47673013647131, 1006.500033578516], [0, 0, 1, 0], [0, 0, 0, 0], [9E9, 9E9, 9E9, 9E9, 9E9, 9E9]];
    CONST robtarget p15059:= [[1469.1632484453567, -56.41355514185693, 1006.500033578516], [0, 0, 1, 0], [0, 0, 0, 0], [9E9, 9E9, 9E9, 9E9, 9E9, 9E9]];
    CONST robtarget p15060:= [[1468.5721818189647, -56.09229880904333, 1006.500033578516], [0, 0, 1, 0], [0, 0, 0, 0], [9E9, 9E9, 9E9, 9E9, 9E9, 9E9]];
    CONST robtarget p15061:= [[1467.787331937398, -55.649631896994535, 1006.500033578516], [0, 0, 1, 0], [0, 0, 0, 0], [9E9, 9E9, 9E9, 9E9, 9E9, 9E9]];
    CONST robtarget p15062:= [[1467.4785234654853, -55.44953024168593, 1006.500033578516], [0, 0, 1, 0], [0, 0, 0, 0], [9E9, 9E9, 9E9, 9E9, 9E9, 9E9]];
    CONST robtarget p15063:= [[1467.050998309803, -55.21453672650589, 1006.500033578516], [0, 0, 1, 0], [0, 0, 0, 0], [9E9, 9E9, 9E9, 9E9, 9E9, 9E9]];
    CONST robtarget p15064:= [[1466.5961163718287, -54.97595999922084, 1006.500033578516], [0, 0, 1, 0], [0, 0, 0, 0], [9E9, 9E9, 9E9, 9E9, 9E9, 9E9]];
    CONST robtarget p15065:= [[1465.9834617962385, -54.59493377964118, 1006.500033578516], [0, 0, 1, 0], [0, 0, 0, 0], [9E9, 9E9, 9E9, 9E9, 9E9, 9E9]];
    CONST robtarget p15066:= [[1465.3800132508347, -54.18240301044895, 1006.500033578516], [0, 0, 1, 0], [0, 0, 0, 0], [9E9, 9E9, 9E9, 9E9, 9E9, 9E9]];
    CONST robtarget p15067:= [[1464.8423044225335, -53.80029592815736, 1006.500033578516], [0, 0, 1, 0], [0, 0, 0, 0], [9E9, 9E9, 9E9, 9E9, 9E9, 9E9]];
    CONST robtarget p15068:= [[1464.7098782516257, -53.71444998937555, 1006.500033578516], [0, 0, 1, 0], [0, 0, 0, 0], [9E9, 9E9, 9E9, 9E9, 9E9, 9E9]];
    CONST robtarget p15069:= [[1464.4361324345443, -53.549152405734986, 1006.500033578516], [0, 0, 1, 0], [0, 0, 0, 0], [9E9, 9E9, 9E9, 9E9, 9E9, 9E9]];
    CONST robtarget p15070:= [[1463.5332132428375, -52.93257690186229, 1006.500033578516], [0, 0, 1, 0], [0, 0, 0, 0], [9E9, 9E9, 9E9, 9E9, 9E9, 9E9]];
    CONST robtarget p15071:= [[1463.3227355983533, -52.80571431446971, 1006.500033578516], [0, 0, 1, 0], [0, 0, 0, 0], [9E9, 9E9, 9E9, 9E9, 9E9, 9E9]];
    CONST robtarget p15072:= [[1462.8089153893777, -52.46703444407636, 1006.500033578516], [0, 0, 1, 0], [0, 0, 0, 0], [9E9, 9E9, 9E9, 9E9, 9E9, 9E9]];
    CONST robtarget p15073:= [[1462.5825761077012, -52.3029725815251, 1006.500033578516], [0, 0, 1, 0], [0, 0, 0, 0], [9E9, 9E9, 9E9, 9E9, 9E9, 9E9]];
    CONST robtarget p15074:= [[1462.1480376195193, -52.017376754393815, 1006.500033578516], [0, 0, 1, 0], [0, 0, 0, 0], [9E9, 9E9, 9E9, 9E9, 9E9, 9E9]];
    CONST robtarget p15075:= [[1461.9832457616799, -51.87514604333668, 1006.500033578516], [0, 0, 1, 0], [0, 0, 0, 0], [9E9, 9E9, 9E9, 9E9, 9E9, 9E9]];
    CONST robtarget p15076:= [[1461.4105508983919, -51.40780363042391, 1006.500033578516], [0, 0, 1, 0], [0, 0, 0, 0], [9E9, 9E9, 9E9, 9E9, 9E9, 9E9]];
    CONST robtarget p15077:= [[1460.820933605111, -50.9905579359953, 1006.500033578516], [0, 0, 1, 0], [0, 0, 0, 0], [9E9, 9E9, 9E9, 9E9, 9E9, 9E9]];
    CONST robtarget p15078:= [[1460.3374392670885, -50.572685488053075, 1006.500033578516], [0, 0, 1, 0], [0, 0, 0, 0], [9E9, 9E9, 9E9, 9E9, 9E9, 9E9]];
    CONST robtarget p15079:= [[1459.773177388402, -50.17387916899156, 1006.500033578516], [0, 0, 1, 0], [0, 0, 0, 0], [9E9, 9E9, 9E9, 9E9, 9E9, 9E9]];
    CONST robtarget p15080:= [[1459.0078211773057, -49.58734578133489, 1006.500033578516], [0, 0, 1, 0], [0, 0, 0, 0], [9E9, 9E9, 9E9, 9E9, 9E9, 9E9]];
    CONST robtarget p15081:= [[1458.4083356034182, -49.01296807765175, 1006.500033578516], [0, 0, 1, 0], [0, 0, 0, 0], [9E9, 9E9, 9E9, 9E9, 9E9, 9E9]];
    CONST robtarget p15082:= [[1458.129098993871, -48.788666644563634, 1006.500033578516], [0, 0, 1, 0], [0, 0, 0, 0], [9E9, 9E9, 9E9, 9E9, 9E9, 9E9]];
    CONST robtarget p15083:= [[1457.8646891736494, -48.58935602497115, 1006.500033578516], [0, 0, 1, 0], [0, 0, 0, 0], [9E9, 9E9, 9E9, 9E9, 9E9, 9E9]];
    CONST robtarget p15084:= [[1457.6666019060597, -48.41312691012406, 1006.500033578516], [0, 0, 1, 0], [0, 0, 0, 0], [9E9, 9E9, 9E9, 9E9, 9E9, 9E9]];
    CONST robtarget p15085:= [[1457.2851112758885, -48.064521017256446, 1006.500033578516], [0, 0, 1, 0], [0, 0, 0, 0], [9E9, 9E9, 9E9, 9E9, 9E9, 9E9]];
    CONST robtarget p15086:= [[1457.163478487681, -47.938522870774065, 1006.500033578516], [0, 0, 1, 0], [0, 0, 0, 0], [9E9, 9E9, 9E9, 9E9, 9E9, 9E9]];
    CONST robtarget p15087:= [[1456.6543731685424, -47.49300515912843, 1006.500033578516], [0, 0, 1, 0], [0, 0, 0, 0], [9E9, 9E9, 9E9, 9E9, 9E9, 9E9]];
    CONST robtarget p15088:= [[1456.1683388414465, -47.05995286433385, 1006.500033578516], [0, 0, 1, 0], [0, 0, 0, 0], [9E9, 9E9, 9E9, 9E9, 9E9, 9E9]];
    CONST robtarget p15089:= [[1455.462484021559, -46.396647011769474, 1006.500033578516], [0, 0, 1, 0], [0, 0, 0, 0], [9E9, 9E9, 9E9, 9E9, 9E9, 9E9]];
    CONST robtarget p15090:= [[1454.6573464845217, -45.61563431995023, 1006.500033578516], [0, 0, 1, 0], [0, 0, 0, 0], [9E9, 9E9, 9E9, 9E9, 9E9, 9E9]];
    CONST robtarget p15091:= [[1454.2817756910508, -45.22102320157401, 1006.500033578516], [0, 0, 1, 0], [0, 0, 0, 0], [9E9, 9E9, 9E9, 9E9, 9E9, 9E9]];
    CONST robtarget p15092:= [[1454.1660991798997, -45.10414992245765, 1006.500033578516], [0, 0, 1, 0], [0, 0, 0, 0], [9E9, 9E9, 9E9, 9E9, 9E9, 9E9]];
    CONST robtarget p15093:= [[1453.9250321865256, -44.862786544789046, 1006.500033578516], [0, 0, 1, 0], [0, 0, 0, 0], [9E9, 9E9, 9E9, 9E9, 9E9, 9E9]];
    CONST robtarget p15094:= [[1453.6496085610866, -44.57271658383445, 1006.500033578516], [0, 0, 1, 0], [0, 0, 0, 0], [9E9, 9E9, 9E9, 9E9, 9E9, 9E9]];
    CONST robtarget p15095:= [[1453.2739174719543, -44.1739484382781, 1006.500033578516], [0, 0, 1, 0], [0, 0, 0, 0], [9E9, 9E9, 9E9, 9E9, 9E9, 9E9]];
    CONST robtarget p15096:= [[1452.8814744018255, -43.76503261520828, 1006.500033578516], [0, 0, 1, 0], [0, 0, 0, 0], [9E9, 9E9, 9E9, 9E9, 9E9, 9E9]];
    CONST robtarget p15097:= [[1452.5247297361502, -43.40756202532697, 1006.500033578516], [0, 0, 1, 0], [0, 0, 0, 0], [9E9, 9E9, 9E9, 9E9, 9E9, 9E9]];
    CONST robtarget p15098:= [[1452.3434528689136, -43.21541214629097, 1006.500033578516], [0, 0, 1, 0], [0, 0, 0, 0], [9E9, 9E9, 9E9, 9E9, 9E9, 9E9]];
    CONST robtarget p15099:= [[1452.0548749458628, -42.90607006726661, 1006.500033578516], [0, 0, 1, 0], [0, 0, 0, 0], [9E9, 9E9, 9E9, 9E9, 9E9, 9E9]];
    CONST robtarget p15100:= [[1451.7238717451205, -42.51202506496327, 1006.500033578516], [0, 0, 1, 0], [0, 0, 0, 0], [9E9, 9E9, 9E9, 9E9, 9E9, 9E9]];
    CONST robtarget p15101:= [[1451.4067517095268, -42.111204748275625, 1006.500033578516], [0, 0, 1, 0], [0, 0, 0, 0], [9E9, 9E9, 9E9, 9E9, 9E9, 9E9]];
    CONST robtarget p15102:= [[1451.082862140116, -41.70744797027065, 1006.500033578516], [0, 0, 1, 0], [0, 0, 0, 0], [9E9, 9E9, 9E9, 9E9, 9E9, 9E9]];
    CONST robtarget p15103:= [[1450.711896396636, -41.28445699140879, 1006.500033578516], [0, 0, 1, 0], [0, 0, 0, 0], [9E9, 9E9, 9E9, 9E9, 9E9, 9E9]];
    CONST robtarget p15104:= [[1450.5811661014259, -41.123487543354614, 1006.500033578516], [0, 0, 1, 0], [0, 0, 0, 0], [9E9, 9E9, 9E9, 9E9, 9E9, 9E9]];
    CONST robtarget p15105:= [[1450.4607972217527, -40.980080508658105, 1006.500033578516], [0, 0, 1, 0], [0, 0, 0, 0], [9E9, 9E9, 9E9, 9E9, 9E9, 9E9]];
    CONST robtarget p15106:= [[1450.3492790952575, -40.85166786758303, 1006.500033578516], [0, 0, 1, 0], [0, 0, 0, 0], [9E9, 9E9, 9E9, 9E9, 9E9, 9E9]];
    CONST robtarget p15107:= [[1450.3294727061796, -40.82552127453619, 1006.500033578516], [0, 0, 1, 0], [0, 0, 0, 0], [9E9, 9E9, 9E9, 9E9, 9E9, 9E9]];
    CONST robtarget p15108:= [[1450.1523792331056, -40.58471409478136, 1006.500033578516], [0, 0, 1, 0], [0, 0, 0, 0], [9E9, 9E9, 9E9, 9E9, 9E9, 9E9]];
    CONST robtarget p15109:= [[1449.6917065464595, -40.05817166020045, 1006.500033578516], [0, 0, 1, 0], [0, 0, 0, 0], [9E9, 9E9, 9E9, 9E9, 9E9, 9E9]];
    CONST robtarget p15110:= [[1449.5084401266545, -39.85721084247146, 1006.500033578516], [0, 0, 1, 0], [0, 0, 0, 0], [9E9, 9E9, 9E9, 9E9, 9E9, 9E9]];
    CONST robtarget p15111:= [[1448.9035467868055, -39.08636514596376, 1006.500033578516], [0, 0, 1, 0], [0, 0, 0, 0], [9E9, 9E9, 9E9, 9E9, 9E9, 9E9]];
    CONST robtarget p15112:= [[1448.7471162477052, -38.86052407898499, 1006.500033578516], [0, 0, 1, 0], [0, 0, 0, 0], [9E9, 9E9, 9E9, 9E9, 9E9, 9E9]];
    CONST robtarget p15113:= [[1448.4241362440068, -38.40779239794572, 1006.500033578516], [0, 0, 1, 0], [0, 0, 0, 0], [9E9, 9E9, 9E9, 9E9, 9E9, 9E9]];
    CONST robtarget p15114:= [[1448.2825188568095, -38.23165052149751, 1006.500033578516], [0, 0, 1, 0], [0, 0, 0, 0], [9E9, 9E9, 9E9, 9E9, 9E9, 9E9]];
    CONST robtarget p15115:= [[1447.8185765013345, -37.51783146945637, 1006.500033578516], [0, 0, 1, 0], [0, 0, 0, 0], [9E9, 9E9, 9E9, 9E9, 9E9, 9E9]];
    CONST robtarget p15116:= [[1447.3731263151556, -36.960012589502774, 1006.500033578516], [0, 0, 1, 0], [0, 0, 0, 0], [9E9, 9E9, 9E9, 9E9, 9E9, 9E9]];
    CONST robtarget p15117:= [[1447.1118934427777, -36.59334379081489, 1006.500033578516], [0, 0, 1, 0], [0, 0, 0, 0], [9E9, 9E9, 9E9, 9E9, 9E9, 9E9]];
    CONST robtarget p15118:= [[1446.984345487822, -36.41538979213295, 1006.500033578516], [0, 0, 1, 0], [0, 0, 0, 0], [9E9, 9E9, 9E9, 9E9, 9E9, 9E9]];
    CONST robtarget p15119:= [[1446.5154735409772, -35.75364362661288, 1006.500033578516], [0, 0, 1, 0], [0, 0, 0, 0], [9E9, 9E9, 9E9, 9E9, 9E9, 9E9]];
    CONST robtarget p15120:= [[1446.4316541018572, -35.61125804928342, 1006.500033578516], [0, 0, 1, 0], [0, 0, 0, 0], [9E9, 9E9, 9E9, 9E9, 9E9, 9E9]];
    CONST robtarget p15121:= [[1446.0936682279716, -35.084124008860485, 1006.500033578516], [0, 0, 1, 0], [0, 0, 0, 0], [9E9, 9E9, 9E9, 9E9, 9E9, 9E9]];
    CONST robtarget p15122:= [[1445.9838671233802, -34.9242604156481, 1006.500033578516], [0, 0, 1, 0], [0, 0, 0, 0], [9E9, 9E9, 9E9, 9E9, 9E9, 9E9]];
    CONST robtarget p15123:= [[1445.863657913446, -34.734717618517934, 1006.500033578516], [0, 0, 1, 0], [0, 0, 0, 0], [9E9, 9E9, 9E9, 9E9, 9E9, 9E9]];
    CONST robtarget p15124:= [[1445.6162174401893, -34.314050489648466, 1006.500033578516], [0, 0, 1, 0], [0, 0, 0, 0], [9E9, 9E9, 9E9, 9E9, 9E9, 9E9]];
    CONST robtarget p15125:= [[1445.092231405861, -33.378316439252494, 1006.500033578516], [0, 0, 1, 0], [0, 0, 0, 0], [9E9, 9E9, 9E9, 9E9, 9E9, 9E9]];
    CONST robtarget p15126:= [[1444.812202289028, -32.98778010859369, 1006.500033578516], [0, 0, 1, 0], [0, 0, 0, 0], [9E9, 9E9, 9E9, 9E9, 9E9, 9E9]];
    CONST robtarget p15127:= [[1444.4586783274679, -32.43015509957643, 1006.500033578516], [0, 0, 1, 0], [0, 0, 0, 0], [9E9, 9E9, 9E9, 9E9, 9E9, 9E9]];
    CONST robtarget p15128:= [[1444.3377457793517, -32.225342956625774, 1006.500033578516], [0, 0, 1, 0], [0, 0, 0, 0], [9E9, 9E9, 9E9, 9E9, 9E9, 9E9]];
    CONST robtarget p15129:= [[1443.9309420100585, -31.544972045904544, 1006.500033578516], [0, 0, 1, 0], [0, 0, 0, 0], [9E9, 9E9, 9E9, 9E9, 9E9, 9E9]];
    CONST robtarget p15130:= [[1443.9248193921103, -31.533404934038444, 1006.500033578516], [0, 0, 1, 0], [0, 0, 0, 0], [9E9, 9E9, 9E9, 9E9, 9E9, 9E9]];
    CONST robtarget p15131:= [[1443.7724590907762, -31.249486255876285, 1006.500033578516], [0, 0, 1, 0], [0, 0, 0, 0], [9E9, 9E9, 9E9, 9E9, 9E9, 9E9]];
    CONST robtarget p15132:= [[1443.6534116016012, -31.01336937396988, 1006.500033578516], [0, 0, 1, 0], [0, 0, 0, 0], [9E9, 9E9, 9E9, 9E9, 9E9, 9E9]];
    CONST robtarget p15133:= [[1443.3587664612653, -30.399550516295434, 1006.500033578516], [0, 0, 1, 0], [0, 0, 0, 0], [9E9, 9E9, 9E9, 9E9, 9E9, 9E9]];
    CONST robtarget p15134:= [[1443.050564728522, -29.861793194226728, 1006.500033578516], [0, 0, 1, 0], [0, 0, 0, 0], [9E9, 9E9, 9E9, 9E9, 9E9, 9E9]];
    CONST robtarget p15135:= [[1442.8070866452726, -29.36082329258886, 1006.500033578516], [0, 0, 1, 0], [0, 0, 0, 0], [9E9, 9E9, 9E9, 9E9, 9E9, 9E9]];
    CONST robtarget p15136:= [[1442.3990211249165, -28.560870190181127, 1006.500033578516], [0, 0, 1, 0], [0, 0, 0, 0], [9E9, 9E9, 9E9, 9E9, 9E9, 9E9]];
    CONST robtarget p15137:= [[1442.2510853993438, -28.287069257814025, 1006.500033578516], [0, 0, 1, 0], [0, 0, 0, 0], [9E9, 9E9, 9E9, 9E9, 9E9, 9E9]];
    CONST robtarget p15138:= [[1441.878586890523, -27.54430418908438, 1006.500033578516], [0, 0, 1, 0], [0, 0, 0, 0], [9E9, 9E9, 9E9, 9E9, 9E9, 9E9]];
    CONST robtarget p15139:= [[1441.688175467527, -27.19852248725841, 1006.500033578516], [0, 0, 1, 0], [0, 0, 0, 0], [9E9, 9E9, 9E9, 9E9, 9E9, 9E9]];
    CONST robtarget p15140:= [[1441.5452109121513, -26.87105094414389, 1006.500033578516], [0, 0, 1, 0], [0, 0, 0, 0], [9E9, 9E9, 9E9, 9E9, 9E9, 9E9]];
    CONST robtarget p15141:= [[1441.2422158860609, -26.06066389357416, 1006.500033578516], [0, 0, 1, 0], [0, 0, 0, 0], [9E9, 9E9, 9E9, 9E9, 9E9, 9E9]];
    CONST robtarget p15142:= [[1441.0675881916034, -25.688108761140548, 1006.500033578516], [0, 0, 1, 0], [0, 0, 0, 0], [9E9, 9E9, 9E9, 9E9, 9E9, 9E9]];
    CONST robtarget p15143:= [[1440.8580391423682, -25.240644220902176, 1006.500033578516], [0, 0, 1, 0], [0, 0, 0, 0], [9E9, 9E9, 9E9, 9E9, 9E9, 9E9]];
    CONST robtarget p15144:= [[1440.835942761683, -25.197969327132682, 1006.500033578516], [0, 0, 1, 0], [0, 0, 0, 0], [9E9, 9E9, 9E9, 9E9, 9E9, 9E9]];
    CONST robtarget p15145:= [[1440.538287581836, -24.486502838938286, 1006.500033578516], [0, 0, 1, 0], [0, 0, 0, 0], [9E9, 9E9, 9E9, 9E9, 9E9, 9E9]];
    CONST robtarget p15146:= [[1440.416254474488, -24.184577034024095, 1006.500033578516], [0, 0, 1, 0], [0, 0, 0, 0], [9E9, 9E9, 9E9, 9E9, 9E9, 9E9]];
    CONST robtarget p15147:= [[1440.1247454613756, -23.430269589289495, 1006.500033578516], [0, 0, 1, 0], [0, 0, 0, 0], [9E9, 9E9, 9E9, 9E9, 9E9, 9E9]];
    CONST robtarget p15148:= [[1439.9409195655717, -23.07998106717369, 1006.500033578516], [0, 0, 1, 0], [0, 0, 0, 0], [9E9, 9E9, 9E9, 9E9, 9E9, 9E9]];
    CONST robtarget p15149:= [[1439.8969661305082, -22.947253418673718, 1006.500033578516], [0, 0, 1, 0], [0, 0, 0, 0], [9E9, 9E9, 9E9, 9E9, 9E9, 9E9]];
    CONST robtarget p15150:= [[1439.7923989985695, -22.584756920511353, 1006.500033578516], [0, 0, 1, 0], [0, 0, 0, 0], [9E9, 9E9, 9E9, 9E9, 9E9, 9E9]];
    CONST robtarget p15151:= [[1439.5619297914839, -21.901882014622814, 1006.500033578516], [0, 0, 1, 0], [0, 0, 0, 0], [9E9, 9E9, 9E9, 9E9, 9E9, 9E9]];
    CONST robtarget p15152:= [[1439.3872095084455, -21.42713688257956, 1006.500033578516], [0, 0, 1, 0], [0, 0, 0, 0], [9E9, 9E9, 9E9, 9E9, 9E9, 9E9]];
    CONST robtarget p15153:= [[1439.3053831809123, -21.232612563056833, 1006.500033578516], [0, 0, 1, 0], [0, 0, 0, 0], [9E9, 9E9, 9E9, 9E9, 9E9, 9E9]];
    CONST robtarget p15154:= [[1439.1844350361303, -20.855242742939033, 1006.500033578516], [0, 0, 1, 0], [0, 0, 0, 0], [9E9, 9E9, 9E9, 9E9, 9E9, 9E9]];
    CONST robtarget p15155:= [[1438.9279993951009, -20.117890717325572, 1006.500033578516], [0, 0, 1, 0], [0, 0, 0, 0], [9E9, 9E9, 9E9, 9E9, 9E9, 9E9]];
    CONST robtarget p15156:= [[1438.8860633288596, -20.01885841689989, 1006.500033578516], [0, 0, 1, 0], [0, 0, 0, 0], [9E9, 9E9, 9E9, 9E9, 9E9, 9E9]];
    CONST robtarget p15157:= [[1438.7993524840447, -19.75203194736867, 1006.500033578516], [0, 0, 1, 0], [0, 0, 0, 0], [9E9, 9E9, 9E9, 9E9, 9E9, 9E9]];
    CONST robtarget p15158:= [[1438.6345706176853, -19.288213958901558, 1006.500033578516], [0, 0, 1, 0], [0, 0, 0, 0], [9E9, 9E9, 9E9, 9E9, 9E9, 9E9]];
    CONST robtarget p15159:= [[1438.4416140531455, -18.70594411132582, 1006.500033578516], [0, 0, 1, 0], [0, 0, 0, 0], [9E9, 9E9, 9E9, 9E9, 9E9, 9E9]];
    CONST robtarget p15160:= [[1438.3419146899564, -18.332027695872732, 1006.500033578516], [0, 0, 1, 0], [0, 0, 0, 0], [9E9, 9E9, 9E9, 9E9, 9E9, 9E9]];
    CONST robtarget p15161:= [[1438.1856069226526, -17.685330167400338, 1006.500033578516], [0, 0, 1, 0], [0, 0, 0, 0], [9E9, 9E9, 9E9, 9E9, 9E9, 9E9]];
    CONST robtarget p15162:= [[1438.1495709060289, -17.5599368166301, 1006.500033578516], [0, 0, 1, 0], [0, 0, 0, 0], [9E9, 9E9, 9E9, 9E9, 9E9, 9E9]];
    CONST robtarget p15163:= [[1438.0916374276496, -17.31801675086612, 1006.500033578516], [0, 0, 1, 0], [0, 0, 0, 0], [9E9, 9E9, 9E9, 9E9, 9E9, 9E9]];
    CONST robtarget p15164:= [[1437.9189174630706, -16.607171888490697, 1006.500033578516], [0, 0, 1, 0], [0, 0, 0, 0], [9E9, 9E9, 9E9, 9E9, 9E9, 9E9]];
    CONST robtarget p15165:= [[1437.8191804678058, -16.26283492163956, 1006.500033578516], [0, 0, 1, 0], [0, 0, 0, 0], [9E9, 9E9, 9E9, 9E9, 9E9, 9E9]];
    CONST robtarget p15166:= [[1437.664629261501, -15.812503025288464, 1006.500033578516], [0, 0, 1, 0], [0, 0, 0, 0], [9E9, 9E9, 9E9, 9E9, 9E9, 9E9]];
    CONST robtarget p15167:= [[1437.6099820344787, -15.561026029739743, 1006.500033578516], [0, 0, 1, 0], [0, 0, 0, 0], [9E9, 9E9, 9E9, 9E9, 9E9, 9E9]];
    CONST robtarget p15168:= [[1437.5583764096482, -15.300342477221875, 1006.500033578516], [0, 0, 1, 0], [0, 0, 0, 0], [9E9, 9E9, 9E9, 9E9, 9E9, 9E9]];
    CONST robtarget p15169:= [[1437.476408943906, -14.921134025614109, 1006.500033578516], [0, 0, 1, 0], [0, 0, 0, 0], [9E9, 9E9, 9E9, 9E9, 9E9, 9E9]];
    CONST robtarget p15170:= [[1437.314657542025, -14.34293109267086, 1006.500033578516], [0, 0, 1, 0], [0, 0, 0, 0], [9E9, 9E9, 9E9, 9E9, 9E9, 9E9]];
    CONST robtarget p15171:= [[1437.1470439331881, -13.736888726374232, 1006.500033578516], [0, 0, 1, 0], [0, 0, 0, 0], [9E9, 9E9, 9E9, 9E9, 9E9, 9E9]];
    CONST robtarget p15172:= [[1437.050464162405, -13.099032160839855, 1006.500033578516], [0, 0, 1, 0], [0, 0, 0, 0], [9E9, 9E9, 9E9, 9E9, 9E9, 9E9]];
    CONST robtarget p15173:= [[1436.9440386792082, -12.568482562851166, 1006.500033578516], [0, 0, 1, 0], [0, 0, 0, 0], [9E9, 9E9, 9E9, 9E9, 9E9, 9E9]];
    CONST robtarget p15174:= [[1436.8700135387455, -12.1235366498831, 1006.500033578516], [0, 0, 1, 0], [0, 0, 0, 0], [9E9, 9E9, 9E9, 9E9, 9E9, 9E9]];
    CONST robtarget p15175:= [[1436.7448220981855, -11.588142243242281, 1006.500033578516], [0, 0, 1, 0], [0, 0, 0, 0], [9E9, 9E9, 9E9, 9E9, 9E9, 9E9]];
    CONST robtarget p15176:= [[1436.5858652647742, -10.703130392757224, 1006.500033578516], [0, 0, 1, 0], [0, 0, 0, 0], [9E9, 9E9, 9E9, 9E9, 9E9, 9E9]];
    CONST robtarget p15177:= [[1436.553275040469, -10.52982743867792, 1006.500033578516], [0, 0, 1, 0], [0, 0, 0, 0], [9E9, 9E9, 9E9, 9E9, 9E9, 9E9]];
    CONST robtarget p15178:= [[1436.5016672263769, -10.154709040348976, 1006.500033578516], [0, 0, 1, 0], [0, 0, 0, 0], [9E9, 9E9, 9E9, 9E9, 9E9, 9E9]];
    CONST robtarget p15179:= [[1436.3423201140556, -9.406737560036326, 1006.500033578516], [0, 0, 1, 0], [0, 0, 0, 0], [9E9, 9E9, 9E9, 9E9, 9E9, 9E9]];
    CONST robtarget p15180:= [[1436.3038282251266, -9.01634582635684, 1006.500033578516], [0, 0, 1, 0], [0, 0, 0, 0], [9E9, 9E9, 9E9, 9E9, 9E9, 9E9]];
    CONST robtarget p15181:= [[1436.2451939169932, -8.515360537414665, 1006.500033578516], [0, 0, 1, 0], [0, 0, 0, 0], [9E9, 9E9, 9E9, 9E9, 9E9, 9E9]];
    CONST robtarget p15182:= [[1436.172850395842, -7.824328868017204, 1006.500033578516], [0, 0, 1, 0], [0, 0, 0, 0], [9E9, 9E9, 9E9, 9E9, 9E9, 9E9]];
    CONST robtarget p15183:= [[1436.096047214864, -7.069659454121435, 1006.500033578516], [0, 0, 1, 0], [0, 0, 0, 0], [9E9, 9E9, 9E9, 9E9, 9E9, 9E9]];
    CONST robtarget p15184:= [[1436.0567438755213, -6.7137099690921005, 1006.500033578516], [0, 0, 1, 0], [0, 0, 0, 0], [9E9, 9E9, 9E9, 9E9, 9E9, 9E9]];
    CONST robtarget p15185:= [[1435.9940030725948, -6.24675439388426, 1006.500033578516], [0, 0, 1, 0], [0, 0, 0, 0], [9E9, 9E9, 9E9, 9E9, 9E9, 9E9]];
    CONST robtarget p15186:= [[1435.9559389790215, -5.9362845936660165, 1006.500033578516], [0, 0, 1, 0], [0, 0, 0, 0], [9E9, 9E9, 9E9, 9E9, 9E9, 9E9]];
    CONST robtarget p15187:= [[1435.8680542920843, -5.105876048989572, 1006.500033578516], [0, 0, 1, 0], [0, 0, 0, 0], [9E9, 9E9, 9E9, 9E9, 9E9, 9E9]];
    CONST robtarget p15188:= [[1435.8467149710032, -4.687341460995839, 1006.500033578516], [0, 0, 1, 0], [0, 0, 0, 0], [9E9, 9E9, 9E9, 9E9, 9E9, 9E9]];
    CONST robtarget p15189:= [[1434.3427428839107, -3.167665761244308, 1007.500033578516], [0, 0, 1, 0], [0, 0, 0, 0], [9E9, 9E9, 9E9, 9E9, 9E9, 9E9]];
    CONST robtarget p15190:= [[1434.309477818703, -2.4459463250571503, 1007.500033578516], [0, 0, 1, 0], [0, 0, 0, 0], [9E9, 9E9, 9E9, 9E9, 9E9, 9E9]];
    CONST robtarget p15191:= [[1434.2237254939334, -1.5062387673312685, 1007.500033578516], [0, 0, 1, 0], [0, 0, 0, 0], [9E9, 9E9, 9E9, 9E9, 9E9, 9E9]];
    CONST robtarget p15192:= [[1434.230430908085, -1.144123112334583, 1007.500033578516], [0, 0, 1, 0], [0, 0, 0, 0], [9E9, 9E9, 9E9, 9E9, 9E9, 9E9]];
    CONST robtarget p15193:= [[1434.219701436293, -0.8893179595577294, 1007.500033578516], [0, 0, 1, 0], [0, 0, 0, 0], [9E9, 9E9, 9E9, 9E9, 9E9, 9E9]];
    CONST robtarget p15194:= [[1434.2137621469237, -0.576887074315195, 1007.500033578516], [0, 0, 1, 0], [0, 0, 0, 0], [9E9, 9E9, 9E9, 9E9, 9E9, 9E9]];
    CONST robtarget p15195:= [[1434.168346959699, 0.01261580792198913, 1007.500033578516], [0, 0, 1, 0], [0, 0, 0, 0], [9E9, 9E9, 9E9, 9E9, 9E9, 9E9]];
    CONST robtarget p15196:= [[1434.1868175983848, 0.572263476699689, 1007.500033578516], [0, 0, 1, 0], [0, 0, 0, 0], [9E9, 9E9, 9E9, 9E9, 9E9, 9E9]];
    CONST robtarget p15197:= [[1434.213676490571, 1.4624329707649508, 1007.500033578516], [0, 0, 1, 0], [0, 0, 0, 0], [9E9, 9E9, 9E9, 9E9, 9E9, 9E9]];
    CONST robtarget p15198:= [[1434.281867283102, 2.8382134123774847, 1007.500033578516], [0, 0, 1, 0], [0, 0, 0, 0], [9E9, 9E9, 9E9, 9E9, 9E9, 9E9]];
    CONST robtarget p15199:= [[1434.2885563983416, 3.1070701615272185, 1007.500033578516], [0, 0, 1, 0], [0, 0, 0, 0], [9E9, 9E9, 9E9, 9E9, 9E9, 9E9]];
    CONST robtarget p15200:= [[1434.2986452076923, 3.836985382333779, 1007.500033578516], [0, 0, 1, 0], [0, 0, 0, 0], [9E9, 9E9, 9E9, 9E9, 9E9, 9E9]];
    CONST robtarget p15201:= [[1434.3458692139761, 4.825637483098959, 1007.500033578516], [0, 0, 1, 0], [0, 0, 0, 0], [9E9, 9E9, 9E9, 9E9, 9E9, 9E9]];
    CONST robtarget p15202:= [[1434.4056389673265, 5.456953799352874, 1007.500033578516], [0, 0, 1, 0], [0, 0, 0, 0], [9E9, 9E9, 9E9, 9E9, 9E9, 9E9]];
    CONST robtarget p15203:= [[1434.485365146132, 5.9118390207715095, 1007.500033578516], [0, 0, 1, 0], [0, 0, 0, 0], [9E9, 9E9, 9E9, 9E9, 9E9, 9E9]];
    CONST robtarget p15204:= [[1434.4928250130174, 5.956840142881177, 1007.500033578516], [0, 0, 1, 0], [0, 0, 0, 0], [9E9, 9E9, 9E9, 9E9, 9E9, 9E9]];
    CONST robtarget p15205:= [[1434.554009647254, 6.314054319819874, 1007.500033578516], [0, 0, 1, 0], [0, 0, 0, 0], [9E9, 9E9, 9E9, 9E9, 9E9, 9E9]];
    CONST robtarget p15206:= [[1434.6281197412638, 6.9778774764614155, 1007.500033578516], [0, 0, 1, 0], [0, 0, 0, 0], [9E9, 9E9, 9E9, 9E9, 9E9, 9E9]];
    CONST robtarget p15207:= [[1434.6322092680093, 7.537634945579697, 1007.500033578516], [0, 0, 1, 0], [0, 0, 0, 0], [9E9, 9E9, 9E9, 9E9, 9E9, 9E9]];
    CONST robtarget p15208:= [[1434.7281002503446, 8.358683588594829, 1007.500033578516], [0, 0, 1, 0], [0, 0, 0, 0], [9E9, 9E9, 9E9, 9E9, 9E9, 9E9]];
    CONST robtarget p15209:= [[1434.8367441830671, 8.87145964955748, 1007.500033578516], [0, 0, 1, 0], [0, 0, 0, 0], [9E9, 9E9, 9E9, 9E9, 9E9, 9E9]];
    CONST robtarget p15210:= [[1434.9198861251389, 9.478713824610026, 1007.500033578516], [0, 0, 1, 0], [0, 0, 0, 0], [9E9, 9E9, 9E9, 9E9, 9E9, 9E9]];
    CONST robtarget p15211:= [[1434.9473903271678, 10.093920511582695, 1007.500033578516], [0, 0, 1, 0], [0, 0, 0, 0], [9E9, 9E9, 9E9, 9E9, 9E9, 9E9]];
    CONST robtarget p15212:= [[1435.1157405723943, 10.999474613810989, 1007.500033578516], [0, 0, 1, 0], [0, 0, 0, 0], [9E9, 9E9, 9E9, 9E9, 9E9, 9E9]];
    CONST robtarget p15213:= [[1435.20148978684, 11.423481957924139, 1007.500033578516], [0, 0, 1, 0], [0, 0, 0, 0], [9E9, 9E9, 9E9, 9E9, 9E9, 9E9]];
    CONST robtarget p15214:= [[1435.3484882590787, 12.233396780607706, 1007.500033578516], [0, 0, 1, 0], [0, 0, 0, 0], [9E9, 9E9, 9E9, 9E9, 9E9, 9E9]];
    CONST robtarget p15215:= [[1435.3845011460496, 12.414405129877878, 1007.500033578516], [0, 0, 1, 0], [0, 0, 0, 0], [9E9, 9E9, 9E9, 9E9, 9E9, 9E9]];
    CONST robtarget p15216:= [[1435.5156275081615, 13.056631806655915, 1007.500033578516], [0, 0, 1, 0], [0, 0, 0, 0], [9E9, 9E9, 9E9, 9E9, 9E9, 9E9]];
    CONST robtarget p15217:= [[1435.553235927471, 13.359891698770923, 1007.500033578516], [0, 0, 1, 0], [0, 0, 0, 0], [9E9, 9E9, 9E9, 9E9, 9E9, 9E9]];
    CONST robtarget p15218:= [[1435.668676986485, 13.955619030874416, 1007.500033578516], [0, 0, 1, 0], [0, 0, 0, 0], [9E9, 9E9, 9E9, 9E9, 9E9, 9E9]];
    CONST robtarget p15219:= [[1435.8655755410944, 14.76170535787152, 1007.500033578516], [0, 0, 1, 0], [0, 0, 0, 0], [9E9, 9E9, 9E9, 9E9, 9E9, 9E9]];
    CONST robtarget p15220:= [[1435.9696294575776, 15.238580357857643, 1007.500033578516], [0, 0, 1, 0], [0, 0, 0, 0], [9E9, 9E9, 9E9, 9E9, 9E9, 9E9]];
    CONST robtarget p15221:= [[1436.1321193530841, 15.784223767135884, 1007.500033578516], [0, 0, 1, 0], [0, 0, 0, 0], [9E9, 9E9, 9E9, 9E9, 9E9, 9E9]];
    CONST robtarget p15222:= [[1436.205732389977, 16.074981266948726, 1007.500033578516], [0, 0, 1, 0], [0, 0, 0, 0], [9E9, 9E9, 9E9, 9E9, 9E9, 9E9]];
    CONST robtarget p15223:= [[1436.584645624436, 17.25690246871943, 1007.500033578516], [0, 0, 1, 0], [0, 0, 0, 0], [9E9, 9E9, 9E9, 9E9, 9E9, 9E9]];
    CONST robtarget p15224:= [[1436.746678035162, 18.185296921176544, 1007.500033578516], [0, 0, 1, 0], [0, 0, 0, 0], [9E9, 9E9, 9E9, 9E9, 9E9, 9E9]];
    CONST robtarget p15225:= [[1436.8058280833286, 18.341009527041322, 1007.500033578516], [0, 0, 1, 0], [0, 0, 0, 0], [9E9, 9E9, 9E9, 9E9, 9E9, 9E9]];
    CONST robtarget p15226:= [[1437.0622971644636, 19.266468504597825, 1007.500033578516], [0, 0, 1, 0], [0, 0, 0, 0], [9E9, 9E9, 9E9, 9E9, 9E9, 9E9]];
    CONST robtarget p15227:= [[1437.2430177207625, 19.81007290200384, 1007.500033578516], [0, 0, 1, 0], [0, 0, 0, 0], [9E9, 9E9, 9E9, 9E9, 9E9, 9E9]];
    CONST robtarget p15228:= [[1437.3720096746788, 20.223253081137045, 1007.500033578516], [0, 0, 1, 0], [0, 0, 0, 0], [9E9, 9E9, 9E9, 9E9, 9E9, 9E9]];
    CONST robtarget p15229:= [[1437.577845648535, 20.820106282602126, 1007.500033578516], [0, 0, 1, 0], [0, 0, 0, 0], [9E9, 9E9, 9E9, 9E9, 9E9, 9E9]];
    CONST robtarget p15230:= [[1437.7724589780894, 21.262703729207573, 1007.500033578516], [0, 0, 1, 0], [0, 0, 0, 0], [9E9, 9E9, 9E9, 9E9, 9E9, 9E9]];
    CONST robtarget p15231:= [[1437.9907886039216, 21.834960181907434, 1007.500033578516], [0, 0, 1, 0], [0, 0, 0, 0], [9E9, 9E9, 9E9, 9E9, 9E9, 9E9]];
    CONST robtarget p15232:= [[1438.0703815933934, 22.097860747872062, 1007.500033578516], [0, 0, 1, 0], [0, 0, 0, 0], [9E9, 9E9, 9E9, 9E9, 9E9, 9E9]];
    CONST robtarget p15233:= [[1438.1523161972045, 22.351269630743914, 1007.500033578516], [0, 0, 1, 0], [0, 0, 0, 0], [9E9, 9E9, 9E9, 9E9, 9E9, 9E9]];
    CONST robtarget p15234:= [[1438.2482686842006, 22.625532995577217, 1007.500033578516], [0, 0, 1, 0], [0, 0, 0, 0], [9E9, 9E9, 9E9, 9E9, 9E9, 9E9]];
    CONST robtarget p15235:= [[1438.4467868364718, 23.28650157833242, 1007.500033578516], [0, 0, 1, 0], [0, 0, 0, 0], [9E9, 9E9, 9E9, 9E9, 9E9, 9E9]];
    CONST robtarget p15236:= [[1438.5698658288932, 23.597569527361443, 1007.500033578516], [0, 0, 1, 0], [0, 0, 0, 0], [9E9, 9E9, 9E9, 9E9, 9E9, 9E9]];
    CONST robtarget p15237:= [[1438.8521857050462, 24.322981344903866, 1007.500033578516], [0, 0, 1, 0], [0, 0, 0, 0], [9E9, 9E9, 9E9, 9E9, 9E9, 9E9]];
    CONST robtarget p15238:= [[1438.9100012754093, 24.455912906499222, 1007.500033578516], [0, 0, 1, 0], [0, 0, 0, 0], [9E9, 9E9, 9E9, 9E9, 9E9, 9E9]];
    CONST robtarget p15239:= [[1439.1248567067582, 24.960750362769687, 1007.500033578516], [0, 0, 1, 0], [0, 0, 0, 0], [9E9, 9E9, 9E9, 9E9, 9E9, 9E9]];
    CONST robtarget p15240:= [[1439.2646996743833, 25.30972209523584, 1007.500033578516], [0, 0, 1, 0], [0, 0, 0, 0], [9E9, 9E9, 9E9, 9E9, 9E9, 9E9]];
    CONST robtarget p15241:= [[1439.4235291636428, 25.700414860386275, 1007.500033578516], [0, 0, 1, 0], [0, 0, 0, 0], [9E9, 9E9, 9E9, 9E9, 9E9, 9E9]];
    CONST robtarget p15242:= [[1439.5921399217666, 26.07448206023433, 1007.500033578516], [0, 0, 1, 0], [0, 0, 0, 0], [9E9, 9E9, 9E9, 9E9, 9E9, 9E9]];
    CONST robtarget p15243:= [[1439.8286586456284, 26.581946169072367, 1007.500033578516], [0, 0, 1, 0], [0, 0, 0, 0], [9E9, 9E9, 9E9, 9E9, 9E9, 9E9]];
    CONST robtarget p15244:= [[1439.9794076464632, 26.97420772784085, 1007.500033578516], [0, 0, 1, 0], [0, 0, 0, 0], [9E9, 9E9, 9E9, 9E9, 9E9, 9E9]];
    CONST robtarget p15245:= [[1440.4108524566698, 27.960288667049326, 1007.500033578516], [0, 0, 1, 0], [0, 0, 0, 0], [9E9, 9E9, 9E9, 9E9, 9E9, 9E9]];
    CONST robtarget p15246:= [[1440.4354283264695, 28.020995533792714, 1007.500033578516], [0, 0, 1, 0], [0, 0, 0, 0], [9E9, 9E9, 9E9, 9E9, 9E9, 9E9]];
    CONST robtarget p15247:= [[1440.5144766905382, 28.210538001845023, 1007.500033578516], [0, 0, 1, 0], [0, 0, 0, 0], [9E9, 9E9, 9E9, 9E9, 9E9, 9E9]];
    CONST robtarget p15248:= [[1440.761779925234, 28.69108805077174, 1007.500033578516], [0, 0, 1, 0], [0, 0, 0, 0], [9E9, 9E9, 9E9, 9E9, 9E9, 9E9]];
    CONST robtarget p15249:= [[1440.934196890657, 29.029700336249846, 1007.500033578516], [0, 0, 1, 0], [0, 0, 0, 0], [9E9, 9E9, 9E9, 9E9, 9E9, 9E9]];
    CONST robtarget p15250:= [[1441.223797339207, 29.584760038396, 1007.500033578516], [0, 0, 1, 0], [0, 0, 0, 0], [9E9, 9E9, 9E9, 9E9, 9E9, 9E9]];
    CONST robtarget p15251:= [[1441.7796057210498, 30.645152207832595, 1007.500033578516], [0, 0, 1, 0], [0, 0, 0, 0], [9E9, 9E9, 9E9, 9E9, 9E9, 9E9]];
    CONST robtarget p15252:= [[1442.031647597698, 31.087080618105517, 1007.500033578516], [0, 0, 1, 0], [0, 0, 0, 0], [9E9, 9E9, 9E9, 9E9, 9E9, 9E9]];
    CONST robtarget p15253:= [[1442.391864637262, 31.836089731168144, 1007.500033578516], [0, 0, 1, 0], [0, 0, 0, 0], [9E9, 9E9, 9E9, 9E9, 9E9, 9E9]];
    CONST robtarget p15254:= [[1442.6746732111803, 32.33865291723902, 1007.500033578516], [0, 0, 1, 0], [0, 0, 0, 0], [9E9, 9E9, 9E9, 9E9, 9E9, 9E9]];
    CONST robtarget p15255:= [[1442.996107104148, 32.88762021268717, 1007.500033578516], [0, 0, 1, 0], [0, 0, 0, 0], [9E9, 9E9, 9E9, 9E9, 9E9, 9E9]];
    CONST robtarget p15256:= [[1443.461967195114, 33.5809432885837, 1007.500033578516], [0, 0, 1, 0], [0, 0, 0, 0], [9E9, 9E9, 9E9, 9E9, 9E9, 9E9]];
    CONST robtarget p15257:= [[1443.7383190274884, 34.08095312093705, 1007.500033578516], [0, 0, 1, 0], [0, 0, 0, 0], [9E9, 9E9, 9E9, 9E9, 9E9, 9E9]];
    CONST robtarget p15258:= [[1443.7652362003332, 34.13074654708285, 1007.500033578516], [0, 0, 1, 0], [0, 0, 0, 0], [9E9, 9E9, 9E9, 9E9, 9E9, 9E9]];
    CONST robtarget p15259:= [[1443.804437097744, 34.20297006648333, 1007.500033578516], [0, 0, 1, 0], [0, 0, 0, 0], [9E9, 9E9, 9E9, 9E9, 9E9, 9E9]];
    CONST robtarget p15260:= [[1444.1333027923247, 34.772077160818554, 1007.500033578516], [0, 0, 1, 0], [0, 0, 0, 0], [9E9, 9E9, 9E9, 9E9, 9E9, 9E9]];
    CONST robtarget p15261:= [[1444.452274919288, 35.28661583984537, 1007.500033578516], [0, 0, 1, 0], [0, 0, 0, 0], [9E9, 9E9, 9E9, 9E9, 9E9, 9E9]];
    CONST robtarget p15262:= [[1444.5693757023598, 35.4786088767255, 1007.500033578516], [0, 0, 1, 0], [0, 0, 0, 0], [9E9, 9E9, 9E9, 9E9, 9E9, 9E9]];
    CONST robtarget p15263:= [[1444.7526872233057, 35.78378543752338, 1007.500033578516], [0, 0, 1, 0], [0, 0, 0, 0], [9E9, 9E9, 9E9, 9E9, 9E9, 9E9]];
    CONST robtarget p15264:= [[1445.303193377113, 36.54502915692174, 1007.500033578516], [0, 0, 1, 0], [0, 0, 0, 0], [9E9, 9E9, 9E9, 9E9, 9E9, 9E9]];
    CONST robtarget p15265:= [[1445.537153703428, 36.92732958561608, 1007.500033578516], [0, 0, 1, 0], [0, 0, 0, 0], [9E9, 9E9, 9E9, 9E9, 9E9, 9E9]];
    CONST robtarget p15266:= [[1445.9809688351183, 37.57265432451351, 1007.500033578516], [0, 0, 1, 0], [0, 0, 0, 0], [9E9, 9E9, 9E9, 9E9, 9E9, 9E9]];
    CONST robtarget p15267:= [[1446.2026929107983, 37.88343532072521, 1007.500033578516], [0, 0, 1, 0], [0, 0, 0, 0], [9E9, 9E9, 9E9, 9E9, 9E9, 9E9]];
    CONST robtarget p15268:= [[1446.3624606637013, 38.09324581753553, 1007.500033578516], [0, 0, 1, 0], [0, 0, 0, 0], [9E9, 9E9, 9E9, 9E9, 9E9, 9E9]];
    CONST robtarget p15269:= [[1446.7325784881373, 38.600745579771385, 1007.500033578516], [0, 0, 1, 0], [0, 0, 0, 0], [9E9, 9E9, 9E9, 9E9, 9E9, 9E9]];
    CONST robtarget p15270:= [[1446.8995220889872, 38.83522613398959, 1007.500033578516], [0, 0, 1, 0], [0, 0, 0, 0], [9E9, 9E9, 9E9, 9E9, 9E9, 9E9]];
    CONST robtarget p15271:= [[1447.0875800559313, 39.12686189244005, 1007.500033578516], [0, 0, 1, 0], [0, 0, 0, 0], [9E9, 9E9, 9E9, 9E9, 9E9, 9E9]];
    CONST robtarget p15272:= [[1447.2226407943647, 39.282444654359765, 1007.500033578516], [0, 0, 1, 0], [0, 0, 0, 0], [9E9, 9E9, 9E9, 9E9, 9E9, 9E9]];
    CONST robtarget p15273:= [[1447.7308095189392, 40.001360734240095, 1007.500033578516], [0, 0, 1, 0], [0, 0, 0, 0], [9E9, 9E9, 9E9, 9E9, 9E9, 9E9]];
    CONST robtarget p15274:= [[1448.011062241634, 40.37058003509199, 1007.500033578516], [0, 0, 1, 0], [0, 0, 0, 0], [9E9, 9E9, 9E9, 9E9, 9E9, 9E9]];
    CONST robtarget p15275:= [[1448.3646283876124, 40.75805616552431, 1007.500033578516], [0, 0, 1, 0], [0, 0, 0, 0], [9E9, 9E9, 9E9, 9E9, 9E9, 9E9]];
    CONST robtarget p15276:= [[1448.948173657698, 41.46948673433637, 1007.500033578516], [0, 0, 1, 0], [0, 0, 0, 0], [9E9, 9E9, 9E9, 9E9, 9E9, 9E9]];
    CONST robtarget p15277:= [[1449.0412744163837, 41.5961779270625, 1007.500033578516], [0, 0, 1, 0], [0, 0, 0, 0], [9E9, 9E9, 9E9, 9E9, 9E9, 9E9]];
    CONST robtarget p15278:= [[1449.5584641413643, 42.24993060154276, 1007.500033578516], [0, 0, 1, 0], [0, 0, 0, 0], [9E9, 9E9, 9E9, 9E9, 9E9, 9E9]];
    CONST robtarget p15279:= [[1450.1122300365394, 42.90538418475731, 1007.500033578516], [0, 0, 1, 0], [0, 0, 0, 0], [9E9, 9E9, 9E9, 9E9, 9E9, 9E9]];
    CONST robtarget p15280:= [[1450.8667857569274, 43.80416038599461, 1007.500033578516], [0, 0, 1, 0], [0, 0, 0, 0], [9E9, 9E9, 9E9, 9E9, 9E9, 9E9]];
    CONST robtarget p15281:= [[1450.928726677971, 43.89805149443447, 1007.500033578516], [0, 0, 1, 0], [0, 0, 0, 0], [9E9, 9E9, 9E9, 9E9, 9E9, 9E9]];
    CONST robtarget p15282:= [[1451.040778348312, 44.01755210753262, 1007.500033578516], [0, 0, 1, 0], [0, 0, 0, 0], [9E9, 9E9, 9E9, 9E9, 9E9, 9E9]];
    CONST robtarget p15283:= [[1451.112267995241, 44.08188730917591, 1007.500033578516], [0, 0, 1, 0], [0, 0, 0, 0], [9E9, 9E9, 9E9, 9E9, 9E9, 9E9]];
    CONST robtarget p15284:= [[1451.6990647809107, 44.667152035898795, 1007.500033578516], [0, 0, 1, 0], [0, 0, 0, 0], [9E9, 9E9, 9E9, 9E9, 9E9, 9E9]];
    CONST robtarget p15285:= [[1451.8260263366203, 44.81994949376947, 1007.500033578516], [0, 0, 1, 0], [0, 0, 0, 0], [9E9, 9E9, 9E9, 9E9, 9E9, 9E9]];
    CONST robtarget p15286:= [[1452.4650838411897, 45.46830297302124, 1007.500033578516], [0, 0, 1, 0], [0, 0, 0, 0], [9E9, 9E9, 9E9, 9E9, 9E9, 9E9]];
    CONST robtarget p15287:= [[1452.7023441894698, 45.731400305179505, 1007.500033578516], [0, 0, 1, 0], [0, 0, 0, 0], [9E9, 9E9, 9E9, 9E9, 9E9, 9E9]];
    CONST robtarget p15288:= [[1453.0453759472387, 46.04652784228996, 1007.500033578516], [0, 0, 1, 0], [0, 0, 0, 0], [9E9, 9E9, 9E9, 9E9, 9E9, 9E9]];
    CONST robtarget p15289:= [[1453.318237242396, 46.335042552458916, 1007.500033578516], [0, 0, 1, 0], [0, 0, 0, 0], [9E9, 9E9, 9E9, 9E9, 9E9, 9E9]];
    CONST robtarget p15290:= [[1453.6780888167257, 46.756385308267554, 1007.500033578516], [0, 0, 1, 0], [0, 0, 0, 0], [9E9, 9E9, 9E9, 9E9, 9E9, 9E9]];
    CONST robtarget p15291:= [[1454.2100368636948, 47.29050899683938, 1007.500033578516], [0, 0, 1, 0], [0, 0, 0, 0], [9E9, 9E9, 9E9, 9E9, 9E9, 9E9]];
    CONST robtarget p15292:= [[1454.7611987689418, 47.784290246015075, 1007.500033578516], [0, 0, 1, 0], [0, 0, 0, 0], [9E9, 9E9, 9E9, 9E9, 9E9, 9E9]];
    CONST robtarget p15293:= [[1454.84938348434, 47.86167653491475, 1007.500033578516], [0, 0, 1, 0], [0, 0, 0, 0], [9E9, 9E9, 9E9, 9E9, 9E9, 9E9]];
    CONST robtarget p15294:= [[1455.3811076103202, 48.343949117799895, 1007.500033578516], [0, 0, 1, 0], [0, 0, 0, 0], [9E9, 9E9, 9E9, 9E9, 9E9, 9E9]];
    CONST robtarget p15295:= [[1455.7245952554135, 48.64198927992986, 1007.500033578516], [0, 0, 1, 0], [0, 0, 0, 0], [9E9, 9E9, 9E9, 9E9, 9E9, 9E9]];
    CONST robtarget p15296:= [[1456.0224413137778, 48.9106496985554, 1007.500033578516], [0, 0, 1, 0], [0, 0, 0, 0], [9E9, 9E9, 9E9, 9E9, 9E9, 9E9]];
    CONST robtarget p15297:= [[1456.3121234485523, 49.180615277342, 1007.500033578516], [0, 0, 1, 0], [0, 0, 0, 0], [9E9, 9E9, 9E9, 9E9, 9E9, 9E9]];
    CONST robtarget p15298:= [[1456.6621647879651, 49.49094791782257, 1007.500033578516], [0, 0, 1, 0], [0, 0, 0, 0], [9E9, 9E9, 9E9, 9E9, 9E9, 9E9]];
    CONST robtarget p15299:= [[1457.0553567634556, 49.858664132685675, 1007.500033578516], [0, 0, 1, 0], [0, 0, 0, 0], [9E9, 9E9, 9E9, 9E9, 9E9, 9E9]];
